(* CODESYS project EPW_3NE_slave.project
   Title: titoloSenza
   Version: 0.0.0.0
   Author: Tecnico3

Project tree, tasks and I/O mapping:
  MyController : TM241CEC24T/U, Schneider Electric, order no. TM241CEC24T/U, version 4.0.6.18
    application Application
      task MAST (cyclic, interval 10 ms, priority 15, watchdog 100 ms x 1) calls P0_Main, Clock_Encoder
      program P0_Main [SFC]: Init_active, ILS_CAN_active
      function block FB_ILS [FBD]
      function block FB_Steppers [FBD]
      Global_VAR/
        global variables GVL
        global variables GVL_HMI
        global variables GVL_IO
        global variables PersistentVars
        global variables GVL_Motion
      Symbols
      Programma/
        program P9_Slave_to_master [ST]
        program P1_Principale [ST]
        program Clock_Encoder [LD]
        program P7_Allarmi [ST]
    DI : Digital Inputs, Schneider Electric, version 4.0.6.18
        settings: IOs Usage = 3075
        input  iwDI_IW0 : WORD  // IW0
        input  Application.Potenza_Attiva : BOOL  // IW0.I4
        input  Application.UM_Abil_Vol : BOOL  // IW0.I5
        input  Application.DI_Unita_10X : BOOL  // IW0.I6
        input  ibDI_IB1 : BYTE  // IB1
    DQ : Digital Outputs, Schneider Electric, version 4.0.6.18
        settings: Outputs Usage = 15
        output Application.Y_sblocco_Carrelli : BOOL  // QW0.Q4
        output Application.Y_sblocco_Pinze : BOOL  // QW0.Q5
        unmapped channels: QW0, QB1
    Counters : Counters, Schneider Electric, version 4.0.6.18
        settings: Instance name = 'Encoder_Volantino'; B input History = 'old=-1 new=1'; A input History = 'old=-1 new=0'; Temporary Instance name = 'Encoder_Volantino'
    Pulse_Generators : Pulse Generators, Schneider Electric, version 4.0.6.18
        settings: Instance name = 'PTO_0'; REF input History = 'old=8 new=10'; B output History = 'old=-1 new=1'; A output History = 'old=-1 new=0'; Temporary Instance name = 'PTO_0'; Instance name = 'PTO_1'; REF input History = 'old=-1 new=11'; B output History = 'old=-1 new=3'; A output History = 'old=-1 new=2'; Temporary Instance name = 'PTO_1'
    Cartridge_1 : Cartridge, Schneider Electric, version 4.0.6.18
    IO_Bus : IO bus - TM3, Schneider Electric, version 4.0.6.18
    COM_Bus : COM bus, Schneider Electric, version 4.0.6.18
    Ethernet_1 : Ethernet Network, Schneider Electric, version 4.0.6.18
      EthernetIP : EthernetIP, Schneider Electric, version 3.3.0.6
          settings: Major Revision for export = 2; old params for export = [100,150,48,48]; CRC of iomapping for export = -17395944
          input  iwEthernetIP_IW0 : WORD  // IW0
          input  modo_regolazioni : BOOL  // IW0.Bit1
          input  Cancella_allarmi : BOOL  // IW0.Bit7
          input  Token : BOOL  // IW0.Bit9
          input  sblocco_carrelli : BOOL  // IW0.Bit11
          input  sblocco_pinze : BOOL  // IW0.Bit12
          input  position_setting : BOOL  // IW0.Bit14
          input  C1_enable : BOOL  // IW1.Bit0
          input  C1_home : BOOL  // IW1.Bit1
          input  C1_position : BOOL  // IW1.Bit2
          input  C1_jog : BOOL  // IW1.Bit3
          input  C1_setpos : BOOL  // IW1.Bit4
          input  C2_enable : BOOL  // IW2.Bit0
          input  C2_home : BOOL  // IW2.Bit1
          input  C2_position : BOOL  // IW2.Bit2
          input  C2_jog : BOOL  // IW2.Bit3
          input  C2_setpos : BOOL  // IW2.Bit4
          input  C3_enable : BOOL  // IW3.Bit0
          input  C3_home : BOOL  // IW3.Bit1
          input  C3_position : BOOL  // IW3.Bit2
          input  C3_jog : BOOL  // IW3.Bit3
          input  C3_setpos : BOOL  // IW3.Bit4
          input  C4_enable : BOOL  // IW4.Bit0
          input  C4_home : BOOL  // IW4.Bit1
          input  C4_position : BOOL  // IW4.Bit2
          input  C4_jog : BOOL  // IW4.Bit3
          input  C4_setpos : BOOL  // IW4.Bit4
          input  Larg_Bracci_enable : BOOL  // IW5.Bit0
          input  Larg_Bracci_home : BOOL  // IW5.Bit1
          input  Larg_Bracci_position : BOOL  // IW5.Bit2
          input  Larg_Bracci_jog : BOOL  // IW5.Bit3
          input  Larg_Bracci_setpos : BOOL  // IW5.Bit4
          input  Pinza_Sx_enable : BOOL  // IW6.Bit0
          input  Pinza_Sx_home : BOOL  // IW6.Bit1
          input  Pinza_Sx_position : BOOL  // IW6.Bit2
          input  Pinza_Sx_jog : BOOL  // IW6.Bit3
          input  Pinza_Sx_setpos : BOOL  // IW6.Bit4
          input  Pinza_Dx_enable : BOOL  // IW7.Bit0
          input  Pinza_Dx_home : BOOL  // IW7.Bit1
          input  Pinza_Dx_position : BOOL  // IW7.Bit2
          input  Pinza_Dx_jog : BOOL  // IW7.Bit3
          input  Pinza_Dx_setpos : BOOL  // IW7.Bit4
          input  iwEthernetIP_IW8 : WORD  // IW8
          input  iwEthernetIP_IW9 : WORD  // IW9
          input  iwEthernetIP_IW10 : WORD  // IW10
          input  iwEthernetIP_IW11 : WORD  // IW11
          input  iwEthernetIP_IW12 : WORD  // IW12
          input  iwEthernetIP_IW13 : WORD  // IW13
          input  iwEthernetIP_IW14 : WORD  // IW14
          input  iwEthernetIP_IW15 : WORD  // IW15
          input  Target_pos_Carrello_1 : WORD  // IW16
          input  Target_pos_Carrello_2 : WORD  // IW17
          input  Target_pos_Carrello_3 : WORD  // IW18
          input  Target_pos_Carrello_4 : WORD  // IW19
          input  Target_pos_Larg_Bracci : WORD  // IW20
          input  Target_pos_Pinza_Sx : WORD  // IW21
          input  Target_pos_Pinza_Dx : WORD  // IW22
          output PB_Abil_Vol : BOOL  // QW0.Bit5
          output Reverse_Token : BOOL  // QW0.Bit9
          output C1_errore : BOOL  // QW1.Bit0
          output C1_referenced : BOOL  // QW1.Bit1
          output C1_done_abs : BOOL  // QW1.Bit2
          output C1_done_home : BOOL  // QW1.Bit3
          output C1_done_mvadd : BOOL  // QW1.Bit4
          output C1_done_setpos : BOOL  // QW1.Bit5
          output C1_in_position : BOOL  // QW1.Bit6
          output C2_errore : BOOL  // QW2.Bit0
          output C2_referenced : BOOL  // QW2.Bit1
          output C2_done_abs : BOOL  // QW2.Bit2
          output C2_done_home : BOOL  // QW2.Bit3
          output C2_done_mvadd : BOOL  // QW2.Bit4
          output C2_done_setpos : BOOL  // QW2.Bit5
          output C2_in_position : BOOL  // QW2.Bit6
          output C3_errore : BOOL  // QW3.Bit0
          output C3_referenced : BOOL  // QW3.Bit1
          output C3_done_abs : BOOL  // QW3.Bit2
          output C3_done_home : BOOL  // QW3.Bit3
          output C3_done_mvadd : BOOL  // QW3.Bit4
          output C3_done_setpos : BOOL  // QW3.Bit5
          output C3_in_position : BOOL  // QW3.Bit6
          output C4_errore : BOOL  // QW4.Bit0
          output C4_referenced : BOOL  // QW4.Bit1
          output C4_done_abs : BOOL  // QW4.Bit2
          output C4_done_home : BOOL  // QW4.Bit3
          output C4_done_mvadd : BOOL  // QW4.Bit4
          output C4_done_setpos : BOOL  // QW4.Bit5
          output C4_in_position : BOOL  // QW4.Bit6
          output L_br_errore : BOOL  // QW5.Bit0
          output L_br_referenced : BOOL  // QW5.Bit1
          output L_br_done_abs : BOOL  // QW5.Bit2
          output L_br_done_home : BOOL  // QW5.Bit3
          output L_br_done_mvadd : BOOL  // QW5.Bit4
          output L_br_done_setpos : BOOL  // QW5.Bit5
          output L_br_in_position : BOOL  // QW5.Bit6
          output Pinza_sx_errore : BOOL  // QW6.Bit0
          output Pinza_sx_referenced : BOOL  // QW6.Bit1
          output Pinza_sx_done_abs : BOOL  // QW6.Bit2
          output Pinza_sx_done_home : BOOL  // QW6.Bit3
          output Pinza_sx_done_mvadd : BOOL  // QW6.Bit4
          output Pinza_sx_done_setpos : BOOL  // QW6.Bit5
          output Pinza_Sx_in_position : BOOL  // QW6.Bit6
          output Pinza_dx_errore : BOOL  // QW7.Bit0
          output Pinza_dx_referenced : BOOL  // QW7.Bit1
          output Pinza_dx_done_abs : BOOL  // QW7.Bit2
          output Pinza_dx_done_home : BOOL  // QW7.Bit3
          output Pinza_dx_done_mvadd : BOOL  // QW7.Bit4
          output Pinza_dx_done_setpos : BOOL  // QW7.Bit5
          output Pinza_Dx_in_position : BOOL  // QW7.Bit6
          output Fault_Carrello_1 : WORD  // QW8
          output Fault_Carrello_2 : WORD  // QW9
          output Fault_Carrello_3 : WORD  // QW10
          output Fault_Carrello_4 : WORD  // QW11
          output Fault_Larg_Bracci : WORD  // QW12
          output Fault_Pinza_Sx : WORD  // QW13
          output Fault_Pinza_Dx : WORD  // QW14
          output Actual_Position_Carrello_1 : WORD  // QW16
          output Actual_Position_Carrello_2 : WORD  // QW17
          output Actual_Position_Carrello_3 : WORD  // QW18
          output Actual_Position_Carrello_4 : WORD  // QW19
          output Actual_Position_Larg_Bracci : WORD  // QW20
          output Actual_Position_Pinza_Sx : WORD  // QW21
          output Actual_Position_Pinza_Dx : WORD  // QW22
          output Actual_Position_Volantino : WORD  // QW23
          unmapped channels: IW1, IW2, IW3, IW4, IW5, IW6, IW7, IW23, QW0, QW1, QW2, QW3, QW4, QW5, QW6, QW7, QW15
    Serial_Line_1 : Serial line, Schneider Electric, version 4.0.6.18
      SoMachine_Network_Manager : SoMachine-Network Manager, Schneider Electric, version 4.0.0.2
    Serial_Line_2 : Serial line, Schneider Electric, version 4.0.6.18
      Modbus_Manager : Modbus Manager, Schneider Electric, version 4.0.0.2
    CAN_1 : CANopen bus, Schneider Electric, version 4.0.6.18
      CANopen_Performance : CANopen Performance, Schneider Electric, order no. 1806, version 3.0.1.24
          settings: ConfigVersion = 50659584
        ILS_Carrello_1 : Lexium ILS, Schneider Electric, order no. 1, version 3.2.1.0
            settings: General Options.Optional Device = TRUE; NODEIDSAVED = 1; SDO Timeout = 1000000; Explicit Deactivate PDOs = FALSE; EXPERTSETTINGS = False; Nodeguarding.Guard Time = 200 ms; Nodeguarding.Life Time Factor = 2; PDO 16#1803.COBID = 16#0481; pdo4_driveCtrl.Subindex = 16#01; pdo4_modeCtrl.Subindex = 16#02; pdo4_Ref16.Subindex = 16#05; pdo4_Ref32.Subindex = 16#06; pdo4_driveStat.Subindex = 16#04; pdo4_modeStat.Subindex = 16#03; pdo4_Act8.Subindex = 16#07; pdo4_Act32.Subindex = 16#08; SDO List.Set Guardtime.Index = 16#100C; SDO List.Set Guardtime.Subindex = 16#00; SDO List.Set Guardtime.Value = 16#000000C8; SDO List.Set Guardtime.Size = 16; SDO List.Set Guardtime.AbortIfError = FALSE; SDO List.Set Guardtime.JumpToLine = FALSE; SDO List.Set Guardtime.Line = 0; SDO List.Set Lifetime.Index = 16#100D; SDO List.Set Lifetime.Subindex = 16#00; SDO List.Set Lifetime.Value = 16#00000002; SDO List.Set Lifetime.Size = 8; SDO List.Set Lifetime.AbortIfError = FALSE; SDO List.Set Lifetime.JumpToLine = FALSE; SDO List.Set Lifetime.Line = 0; SDO List.Disable PDO.Index = 16#1803; SDO List.Disable PDO.Subindex = 16#01; SDO List.Disable PDO.Value = 16#80000481; SDO List.Disable PDO.Size = 32; SDO List.Disable PDO.AbortIfError = FALSE; SDO List.Disable PDO.JumpToLine = FALSE; SDO List.Disable PDO.Line = 0; SDO List.Set transmission type.Index = 16#1803; SDO List.Set transmission type.Subindex = 16#02; SDO List.Set transmission type.Value = 16#FE;
              SDO List.Set transmission type.Size = 8; SDO List.Set transmission type.AbortIfError = FALSE; SDO List.Set transmission type.JumpToLine = FALSE; SDO List.Set transmission type.Line = 0; SDO List.Set inhibit time.Index = 16#1803; SDO List.Set inhibit time.Subindex = 16#03; SDO List.Set inhibit time.Value = 16#0064; SDO List.Set inhibit time.Size = 16; SDO List.Set inhibit time.AbortIfError = FALSE; SDO List.Set inhibit time.JumpToLine = FALSE; SDO List.Set inhibit time.Line = 0; SDO List.Set event time.Index = 16#1803; SDO List.Set event time.Subindex = 16#05; SDO List.Set event time.Value = 16#0000; SDO List.Set event time.Size = 16; SDO List.Set event time.AbortIfError = FALSE; SDO List.Set event time.JumpToLine = FALSE; SDO List.Set event time.Line = 0; SDO List.Set and enable COB-ID.Index = 16#1803; SDO List.Set and enable COB-ID.Subindex = 16#01; SDO List.Set and enable COB-ID.Value = 16#00000481; SDO List.Set and enable COB-ID.Size = 32; SDO List.Set and enable COB-ID.AbortIfError = FALSE; SDO List.Set and enable COB-ID.JumpToLine = FALSE; SDO List.Set and enable COB-ID.Line = 0; SDO List.Automap SDO1.Index = 16#301E; SDO List.Automap SDO1.Subindex = 16#0A; SDO List.Automap SDO1.Value = 4294967295; SDO List.Automap SDO1.Size = 32; SDO List.Automap SDO1.AbortIfError = FALSE; SDO List.Automap SDO1.JumpToLine = FALSE; SDO List.Automap SDO1.Line = 0; ConfigVersion = 50659584
            unmapped channels: pdo4_driveCtrl, pdo4_modeCtrl, pdo4_Ref16, pdo4_Ref32, pdo4_driveStat, pdo4_modeStat, pdo4_Act8, pdo4_Act32
        ILS_Carrello_2 : Lexium ILS, Schneider Electric, order no. 1, version 3.2.1.0
            settings: General Options.Optional Device = TRUE; NODEIDSAVED = 2; SDO Timeout = 1000000; Explicit Deactivate PDOs = FALSE; EXPERTSETTINGS = FALSE; Nodeguarding.Guard Time = 200 ms; Nodeguarding.Life Time Factor = 2; Emergency-General Parameters.Emergency COBID = 16#82; PDO 16#1403.COBID = 16#40000502; PDO 16#1803.COBID = 16#0482; pdo4_driveCtrl.Subindex = 16#01; pdo4_modeCtrl.Subindex = 16#02; pdo4_Ref16.Subindex = 16#05; pdo4_Ref32.Subindex = 16#06; pdo4_driveStat.Subindex = 16#04; pdo4_modeStat.Subindex = 16#03; pdo4_Act8.Subindex = 16#07; pdo4_Act32.Subindex = 16#08; SDO List.Set Guardtime.Index = 16#100C; SDO List.Set Guardtime.Subindex = 16#00; SDO List.Set Guardtime.Value = 16#000000C8; SDO List.Set Guardtime.Size = 16; SDO List.Set Guardtime.AbortIfError = FALSE; SDO List.Set Guardtime.JumpToLine = FALSE; SDO List.Set Guardtime.Line = 0; SDO List.Set Lifetime.Index = 16#100D; SDO List.Set Lifetime.Subindex = 16#00; SDO List.Set Lifetime.Value = 16#00000002; SDO List.Set Lifetime.Size = 8; SDO List.Set Lifetime.AbortIfError = FALSE; SDO List.Set Lifetime.JumpToLine = FALSE; SDO List.Set Lifetime.Line = 0; SDO List.Disable PDO.Index = 16#1803; SDO List.Disable PDO.Subindex = 16#01; SDO List.Disable PDO.Value = 16#80000482; SDO List.Disable PDO.Size = 32; SDO List.Disable PDO.AbortIfError = FALSE; SDO List.Disable PDO.JumpToLine = FALSE; SDO List.Disable PDO.Line = 0; SDO List.Set transmission type.Index = 16#1803;
              SDO List.Set transmission type.Subindex = 16#02; SDO List.Set transmission type.Value = 16#FE; SDO List.Set transmission type.Size = 8; SDO List.Set transmission type.AbortIfError = FALSE; SDO List.Set transmission type.JumpToLine = FALSE; SDO List.Set transmission type.Line = 0; SDO List.Set inhibit time.Index = 16#1803; SDO List.Set inhibit time.Subindex = 16#03; SDO List.Set inhibit time.Value = 16#0064; SDO List.Set inhibit time.Size = 16; SDO List.Set inhibit time.AbortIfError = FALSE; SDO List.Set inhibit time.JumpToLine = FALSE; SDO List.Set inhibit time.Line = 0; SDO List.Set event time.Index = 16#1803; SDO List.Set event time.Subindex = 16#05; SDO List.Set event time.Value = 16#0000; SDO List.Set event time.Size = 16; SDO List.Set event time.AbortIfError = FALSE; SDO List.Set event time.JumpToLine = FALSE; SDO List.Set event time.Line = 0; SDO List.Set and enable COB-ID.Index = 16#1803; SDO List.Set and enable COB-ID.Subindex = 16#01; SDO List.Set and enable COB-ID.Value = 16#00000482; SDO List.Set and enable COB-ID.Size = 32; SDO List.Set and enable COB-ID.AbortIfError = FALSE; SDO List.Set and enable COB-ID.JumpToLine = FALSE; SDO List.Set and enable COB-ID.Line = 0; SDO List.Automap SDO1.Index = 16#301E; SDO List.Automap SDO1.Subindex = 16#0A; SDO List.Automap SDO1.Value = 4294967295; SDO List.Automap SDO1.Size = 32; SDO List.Automap SDO1.AbortIfError = FALSE; SDO List.Automap SDO1.JumpToLine = FALSE; SDO List.Automap SDO1.Line = 0; ConfigVersion = 50659584
            unmapped channels: pdo4_driveCtrl, pdo4_modeCtrl, pdo4_Ref16, pdo4_Ref32, pdo4_driveStat, pdo4_modeStat, pdo4_Act8, pdo4_Act32
        ILS_Carrello_3 : Lexium ILS, Schneider Electric, order no. 1, version 3.2.1.0
            settings: General Options.Optional Device = TRUE; NODEIDSAVED = 3; SDO Timeout = 1000000; Explicit Deactivate PDOs = FALSE; EXPERTSETTINGS = FALSE; Nodeguarding.Guard Time = 200 ms; Nodeguarding.Life Time Factor = 2; Emergency-General Parameters.Emergency COBID = 16#83; PDO 16#1403.COBID = 16#40000503; PDO 16#1803.COBID = 16#0483; pdo4_driveCtrl.Subindex = 16#01; pdo4_modeCtrl.Subindex = 16#02; pdo4_Ref16.Subindex = 16#05; pdo4_Ref32.Subindex = 16#06; pdo4_driveStat.Subindex = 16#04; pdo4_modeStat.Subindex = 16#03; pdo4_Act8.Subindex = 16#07; pdo4_Act32.Subindex = 16#08; SDO List.Set Guardtime.Index = 16#100C; SDO List.Set Guardtime.Subindex = 16#00; SDO List.Set Guardtime.Value = 16#000000C8; SDO List.Set Guardtime.Size = 16; SDO List.Set Guardtime.AbortIfError = FALSE; SDO List.Set Guardtime.JumpToLine = FALSE; SDO List.Set Guardtime.Line = 0; SDO List.Set Lifetime.Index = 16#100D; SDO List.Set Lifetime.Subindex = 16#00; SDO List.Set Lifetime.Value = 16#00000002; SDO List.Set Lifetime.Size = 8; SDO List.Set Lifetime.AbortIfError = FALSE; SDO List.Set Lifetime.JumpToLine = FALSE; SDO List.Set Lifetime.Line = 0; SDO List.Disable PDO.Index = 16#1803; SDO List.Disable PDO.Subindex = 16#01; SDO List.Disable PDO.Value = 16#80000483; SDO List.Disable PDO.Size = 32; SDO List.Disable PDO.AbortIfError = FALSE; SDO List.Disable PDO.JumpToLine = FALSE; SDO List.Disable PDO.Line = 0; SDO List.Set transmission type.Index = 16#1803;
              SDO List.Set transmission type.Subindex = 16#02; SDO List.Set transmission type.Value = 16#FE; SDO List.Set transmission type.Size = 8; SDO List.Set transmission type.AbortIfError = FALSE; SDO List.Set transmission type.JumpToLine = FALSE; SDO List.Set transmission type.Line = 0; SDO List.Set inhibit time.Index = 16#1803; SDO List.Set inhibit time.Subindex = 16#03; SDO List.Set inhibit time.Value = 16#0064; SDO List.Set inhibit time.Size = 16; SDO List.Set inhibit time.AbortIfError = FALSE; SDO List.Set inhibit time.JumpToLine = FALSE; SDO List.Set inhibit time.Line = 0; SDO List.Set event time.Index = 16#1803; SDO List.Set event time.Subindex = 16#05; SDO List.Set event time.Value = 16#0000; SDO List.Set event time.Size = 16; SDO List.Set event time.AbortIfError = FALSE; SDO List.Set event time.JumpToLine = FALSE; SDO List.Set event time.Line = 0; SDO List.Set and enable COB-ID.Index = 16#1803; SDO List.Set and enable COB-ID.Subindex = 16#01; SDO List.Set and enable COB-ID.Value = 16#00000483; SDO List.Set and enable COB-ID.Size = 32; SDO List.Set and enable COB-ID.AbortIfError = FALSE; SDO List.Set and enable COB-ID.JumpToLine = FALSE; SDO List.Set and enable COB-ID.Line = 0; SDO List.Automap SDO1.Index = 16#301E; SDO List.Automap SDO1.Subindex = 16#0A; SDO List.Automap SDO1.Value = 4294967295; SDO List.Automap SDO1.Size = 32; SDO List.Automap SDO1.AbortIfError = FALSE; SDO List.Automap SDO1.JumpToLine = FALSE; SDO List.Automap SDO1.Line = 0; ConfigVersion = 50659584
            unmapped channels: pdo4_driveCtrl, pdo4_modeCtrl, pdo4_Ref16, pdo4_Ref32, pdo4_driveStat, pdo4_modeStat, pdo4_Act8, pdo4_Act32
        ILS_Carrello_4 : Lexium ILS, Schneider Electric, order no. 1, version 3.2.1.0
            settings: General Options.Optional Device = TRUE; NODEIDSAVED = 4; SDO Timeout = 1000000; Explicit Deactivate PDOs = FALSE; EXPERTSETTINGS = FALSE; Nodeguarding.Guard Time = 200 ms; Nodeguarding.Life Time Factor = 2; Emergency-General Parameters.Emergency COBID = 16#84; PDO 16#1403.COBID = 16#40000504; PDO 16#1803.COBID = 16#0484; pdo4_driveCtrl.Subindex = 16#01; pdo4_modeCtrl.Subindex = 16#02; pdo4_Ref16.Subindex = 16#05; pdo4_Ref32.Subindex = 16#06; pdo4_driveStat.Subindex = 16#04; pdo4_modeStat.Subindex = 16#03; pdo4_Act8.Subindex = 16#07; pdo4_Act32.Subindex = 16#08; SDO List.Set Guardtime.Index = 16#100C; SDO List.Set Guardtime.Subindex = 16#00; SDO List.Set Guardtime.Value = 16#000000C8; SDO List.Set Guardtime.Size = 16; SDO List.Set Guardtime.AbortIfError = FALSE; SDO List.Set Guardtime.JumpToLine = FALSE; SDO List.Set Guardtime.Line = 0; SDO List.Set Lifetime.Index = 16#100D; SDO List.Set Lifetime.Subindex = 16#00; SDO List.Set Lifetime.Value = 16#00000002; SDO List.Set Lifetime.Size = 8; SDO List.Set Lifetime.AbortIfError = FALSE; SDO List.Set Lifetime.JumpToLine = FALSE; SDO List.Set Lifetime.Line = 0; SDO List.Disable PDO.Index = 16#1803; SDO List.Disable PDO.Subindex = 16#01; SDO List.Disable PDO.Value = 16#80000484; SDO List.Disable PDO.Size = 32; SDO List.Disable PDO.AbortIfError = FALSE; SDO List.Disable PDO.JumpToLine = FALSE; SDO List.Disable PDO.Line = 0; SDO List.Set transmission type.Index = 16#1803;
              SDO List.Set transmission type.Subindex = 16#02; SDO List.Set transmission type.Value = 16#FE; SDO List.Set transmission type.Size = 8; SDO List.Set transmission type.AbortIfError = FALSE; SDO List.Set transmission type.JumpToLine = FALSE; SDO List.Set transmission type.Line = 0; SDO List.Set inhibit time.Index = 16#1803; SDO List.Set inhibit time.Subindex = 16#03; SDO List.Set inhibit time.Value = 16#0064; SDO List.Set inhibit time.Size = 16; SDO List.Set inhibit time.AbortIfError = FALSE; SDO List.Set inhibit time.JumpToLine = FALSE; SDO List.Set inhibit time.Line = 0; SDO List.Set event time.Index = 16#1803; SDO List.Set event time.Subindex = 16#05; SDO List.Set event time.Value = 16#0000; SDO List.Set event time.Size = 16; SDO List.Set event time.AbortIfError = FALSE; SDO List.Set event time.JumpToLine = FALSE; SDO List.Set event time.Line = 0; SDO List.Set and enable COB-ID.Index = 16#1803; SDO List.Set and enable COB-ID.Subindex = 16#01; SDO List.Set and enable COB-ID.Value = 16#00000484; SDO List.Set and enable COB-ID.Size = 32; SDO List.Set and enable COB-ID.AbortIfError = FALSE; SDO List.Set and enable COB-ID.JumpToLine = FALSE; SDO List.Set and enable COB-ID.Line = 0; SDO List.Automap SDO1.Index = 16#301E; SDO List.Automap SDO1.Subindex = 16#0A; SDO List.Automap SDO1.Value = 4294967295; SDO List.Automap SDO1.Size = 32; SDO List.Automap SDO1.AbortIfError = FALSE; SDO List.Automap SDO1.JumpToLine = FALSE; SDO List.Automap SDO1.Line = 0; ConfigVersion = 50659584
            unmapped channels: pdo4_driveCtrl, pdo4_modeCtrl, pdo4_Ref16, pdo4_Ref32, pdo4_driveStat, pdo4_modeStat, pdo4_Act8, pdo4_Act32
        ILS_Larg_Bracci : Lexium ILS, Schneider Electric, order no. 1, version 3.2.1.0
            settings: General Options.Optional Device = TRUE; NODEIDSAVED = 5; SDO Timeout = 1000000; Explicit Deactivate PDOs = FALSE; EXPERTSETTINGS = FALSE; Nodeguarding.Guard Time = 200 ms; Nodeguarding.Life Time Factor = 2; Emergency-General Parameters.Emergency COBID = 16#85; PDO 16#1403.COBID = 16#40000505; PDO 16#1803.COBID = 16#0485; pdo4_driveCtrl.Subindex = 16#01; pdo4_modeCtrl.Subindex = 16#02; pdo4_Ref16.Subindex = 16#05; pdo4_Ref32.Subindex = 16#06; pdo4_driveStat.Subindex = 16#04; pdo4_modeStat.Subindex = 16#03; pdo4_Act8.Subindex = 16#07; pdo4_Act32.Subindex = 16#08; SDO List.Set Guardtime.Index = 16#100C; SDO List.Set Guardtime.Subindex = 16#00; SDO List.Set Guardtime.Value = 16#000000C8; SDO List.Set Guardtime.Size = 16; SDO List.Set Guardtime.AbortIfError = FALSE; SDO List.Set Guardtime.JumpToLine = FALSE; SDO List.Set Guardtime.Line = 0; SDO List.Set Lifetime.Index = 16#100D; SDO List.Set Lifetime.Subindex = 16#00; SDO List.Set Lifetime.Value = 16#00000002; SDO List.Set Lifetime.Size = 8; SDO List.Set Lifetime.AbortIfError = FALSE; SDO List.Set Lifetime.JumpToLine = FALSE; SDO List.Set Lifetime.Line = 0; SDO List.Disable PDO.Index = 16#1803; SDO List.Disable PDO.Subindex = 16#01; SDO List.Disable PDO.Value = 16#80000485; SDO List.Disable PDO.Size = 32; SDO List.Disable PDO.AbortIfError = FALSE; SDO List.Disable PDO.JumpToLine = FALSE; SDO List.Disable PDO.Line = 0; SDO List.Set transmission type.Index = 16#1803;
              SDO List.Set transmission type.Subindex = 16#02; SDO List.Set transmission type.Value = 16#FE; SDO List.Set transmission type.Size = 8; SDO List.Set transmission type.AbortIfError = FALSE; SDO List.Set transmission type.JumpToLine = FALSE; SDO List.Set transmission type.Line = 0; SDO List.Set inhibit time.Index = 16#1803; SDO List.Set inhibit time.Subindex = 16#03; SDO List.Set inhibit time.Value = 16#0064; SDO List.Set inhibit time.Size = 16; SDO List.Set inhibit time.AbortIfError = FALSE; SDO List.Set inhibit time.JumpToLine = FALSE; SDO List.Set inhibit time.Line = 0; SDO List.Set event time.Index = 16#1803; SDO List.Set event time.Subindex = 16#05; SDO List.Set event time.Value = 16#0000; SDO List.Set event time.Size = 16; SDO List.Set event time.AbortIfError = FALSE; SDO List.Set event time.JumpToLine = FALSE; SDO List.Set event time.Line = 0; SDO List.Set and enable COB-ID.Index = 16#1803; SDO List.Set and enable COB-ID.Subindex = 16#01; SDO List.Set and enable COB-ID.Value = 16#00000485; SDO List.Set and enable COB-ID.Size = 32; SDO List.Set and enable COB-ID.AbortIfError = FALSE; SDO List.Set and enable COB-ID.JumpToLine = FALSE; SDO List.Set and enable COB-ID.Line = 0; SDO List.Automap SDO1.Index = 16#301E; SDO List.Automap SDO1.Subindex = 16#0A; SDO List.Automap SDO1.Value = 4294967295; SDO List.Automap SDO1.Size = 32; SDO List.Automap SDO1.AbortIfError = FALSE; SDO List.Automap SDO1.JumpToLine = FALSE; SDO List.Automap SDO1.Line = 0; ConfigVersion = 50659584
            unmapped channels: pdo4_driveCtrl, pdo4_modeCtrl, pdo4_Ref16, pdo4_Ref32, pdo4_driveStat, pdo4_modeStat, pdo4_Act8, pdo4_Act32
        ILS_Pinza_Sx : Lexium ILS, Schneider Electric, order no. 1, version 3.2.1.0
            settings: General Options.Optional Device = TRUE; NODEIDSAVED = 6; SDO Timeout = 1000000; Explicit Deactivate PDOs = FALSE; EXPERTSETTINGS = FALSE; Nodeguarding.Guard Time = 200 ms; Nodeguarding.Life Time Factor = 2; Emergency-General Parameters.Emergency COBID = 16#86; PDO 16#1403.COBID = 16#40000506; PDO 16#1803.COBID = 16#0486; pdo4_driveCtrl.Subindex = 16#01; pdo4_modeCtrl.Subindex = 16#02; pdo4_Ref16.Subindex = 16#05; pdo4_Ref32.Subindex = 16#06; pdo4_driveStat.Subindex = 16#04; pdo4_modeStat.Subindex = 16#03; pdo4_Act8.Subindex = 16#07; pdo4_Act32.Subindex = 16#08; SDO List.Set Guardtime.Index = 16#100C; SDO List.Set Guardtime.Subindex = 16#00; SDO List.Set Guardtime.Value = 16#000000C8; SDO List.Set Guardtime.Size = 16; SDO List.Set Guardtime.AbortIfError = FALSE; SDO List.Set Guardtime.JumpToLine = FALSE; SDO List.Set Guardtime.Line = 0; SDO List.Set Lifetime.Index = 16#100D; SDO List.Set Lifetime.Subindex = 16#00; SDO List.Set Lifetime.Value = 16#00000002; SDO List.Set Lifetime.Size = 8; SDO List.Set Lifetime.AbortIfError = FALSE; SDO List.Set Lifetime.JumpToLine = FALSE; SDO List.Set Lifetime.Line = 0; SDO List.Disable PDO.Index = 16#1803; SDO List.Disable PDO.Subindex = 16#01; SDO List.Disable PDO.Value = 16#80000486; SDO List.Disable PDO.Size = 32; SDO List.Disable PDO.AbortIfError = FALSE; SDO List.Disable PDO.JumpToLine = FALSE; SDO List.Disable PDO.Line = 0; SDO List.Set transmission type.Index = 16#1803;
              SDO List.Set transmission type.Subindex = 16#02; SDO List.Set transmission type.Value = 16#FE; SDO List.Set transmission type.Size = 8; SDO List.Set transmission type.AbortIfError = FALSE; SDO List.Set transmission type.JumpToLine = FALSE; SDO List.Set transmission type.Line = 0; SDO List.Set inhibit time.Index = 16#1803; SDO List.Set inhibit time.Subindex = 16#03; SDO List.Set inhibit time.Value = 16#0064; SDO List.Set inhibit time.Size = 16; SDO List.Set inhibit time.AbortIfError = FALSE; SDO List.Set inhibit time.JumpToLine = FALSE; SDO List.Set inhibit time.Line = 0; SDO List.Set event time.Index = 16#1803; SDO List.Set event time.Subindex = 16#05; SDO List.Set event time.Value = 16#0000; SDO List.Set event time.Size = 16; SDO List.Set event time.AbortIfError = FALSE; SDO List.Set event time.JumpToLine = FALSE; SDO List.Set event time.Line = 0; SDO List.Set and enable COB-ID.Index = 16#1803; SDO List.Set and enable COB-ID.Subindex = 16#01; SDO List.Set and enable COB-ID.Value = 16#00000486; SDO List.Set and enable COB-ID.Size = 32; SDO List.Set and enable COB-ID.AbortIfError = FALSE; SDO List.Set and enable COB-ID.JumpToLine = FALSE; SDO List.Set and enable COB-ID.Line = 0; SDO List.Automap SDO1.Index = 16#301E; SDO List.Automap SDO1.Subindex = 16#0A; SDO List.Automap SDO1.Value = 4294967295; SDO List.Automap SDO1.Size = 32; SDO List.Automap SDO1.AbortIfError = FALSE; SDO List.Automap SDO1.JumpToLine = FALSE; SDO List.Automap SDO1.Line = 0; ConfigVersion = 50659584
            unmapped channels: pdo4_driveCtrl, pdo4_modeCtrl, pdo4_Ref16, pdo4_Ref32, pdo4_driveStat, pdo4_modeStat, pdo4_Act8, pdo4_Act32
        ILS_Pinza_Dx : Lexium ILS, Schneider Electric, order no. 1, version 3.2.1.0
            settings: General Options.Optional Device = TRUE; NODEIDSAVED = 7; SDO Timeout = 1000000; Explicit Deactivate PDOs = FALSE; EXPERTSETTINGS = FALSE; Nodeguarding.Guard Time = 200 ms; Nodeguarding.Life Time Factor = 2; Emergency-General Parameters.Emergency COBID = 16#87; PDO 16#1403.COBID = 16#40000507; PDO 16#1803.COBID = 16#0487; pdo4_driveCtrl.Subindex = 16#01; pdo4_modeCtrl.Subindex = 16#02; pdo4_Ref16.Subindex = 16#05; pdo4_Ref32.Subindex = 16#06; pdo4_driveStat.Subindex = 16#04; pdo4_modeStat.Subindex = 16#03; pdo4_Act8.Subindex = 16#07; pdo4_Act32.Subindex = 16#08; SDO List.Set Guardtime.Index = 16#100C; SDO List.Set Guardtime.Subindex = 16#00; SDO List.Set Guardtime.Value = 16#000000C8; SDO List.Set Guardtime.Size = 16; SDO List.Set Guardtime.AbortIfError = FALSE; SDO List.Set Guardtime.JumpToLine = FALSE; SDO List.Set Guardtime.Line = 0; SDO List.Set Lifetime.Index = 16#100D; SDO List.Set Lifetime.Subindex = 16#00; SDO List.Set Lifetime.Value = 16#00000002; SDO List.Set Lifetime.Size = 8; SDO List.Set Lifetime.AbortIfError = FALSE; SDO List.Set Lifetime.JumpToLine = FALSE; SDO List.Set Lifetime.Line = 0; SDO List.Disable PDO.Index = 16#1803; SDO List.Disable PDO.Subindex = 16#01; SDO List.Disable PDO.Value = 16#80000487; SDO List.Disable PDO.Size = 32; SDO List.Disable PDO.AbortIfError = FALSE; SDO List.Disable PDO.JumpToLine = FALSE; SDO List.Disable PDO.Line = 0; SDO List.Set transmission type.Index = 16#1803;
              SDO List.Set transmission type.Subindex = 16#02; SDO List.Set transmission type.Value = 16#FE; SDO List.Set transmission type.Size = 8; SDO List.Set transmission type.AbortIfError = FALSE; SDO List.Set transmission type.JumpToLine = FALSE; SDO List.Set transmission type.Line = 0; SDO List.Set inhibit time.Index = 16#1803; SDO List.Set inhibit time.Subindex = 16#03; SDO List.Set inhibit time.Value = 16#0064; SDO List.Set inhibit time.Size = 16; SDO List.Set inhibit time.AbortIfError = FALSE; SDO List.Set inhibit time.JumpToLine = FALSE; SDO List.Set inhibit time.Line = 0; SDO List.Set event time.Index = 16#1803; SDO List.Set event time.Subindex = 16#05; SDO List.Set event time.Value = 16#0000; SDO List.Set event time.Size = 16; SDO List.Set event time.AbortIfError = FALSE; SDO List.Set event time.JumpToLine = FALSE; SDO List.Set event time.Line = 0; SDO List.Set and enable COB-ID.Index = 16#1803; SDO List.Set and enable COB-ID.Subindex = 16#01; SDO List.Set and enable COB-ID.Value = 16#00000487; SDO List.Set and enable COB-ID.Size = 32; SDO List.Set and enable COB-ID.AbortIfError = FALSE; SDO List.Set and enable COB-ID.JumpToLine = FALSE; SDO List.Set and enable COB-ID.Line = 0; SDO List.Automap SDO1.Index = 16#301E; SDO List.Automap SDO1.Subindex = 16#0A; SDO List.Automap SDO1.Value = 4294967295; SDO List.Automap SDO1.Size = 32; SDO List.Automap SDO1.AbortIfError = FALSE; SDO List.Automap SDO1.JumpToLine = FALSE; SDO List.Automap SDO1.Line = 0; ConfigVersion = 50659584
            unmapped channels: pdo4_driveCtrl, pdo4_modeCtrl, pdo4_Ref16, pdo4_Ref32, pdo4_driveStat, pdo4_modeStat, pdo4_Act8, pdo4_Act32
*)

// MyController/Application/Global_VAR/GVL
VAR_GLOBAL
	Power_Carrello_1: BOOL;
	Stop_Carrello_1: BOOL;
	Reset_Carrello_1: BOOL;
	Home_Carrello_1: BOOL;
	Home_Pos_Carrello_1: DINT;
	HomingMode_Carrello_1: UINT;
	VHome_Carrello_1: UINT;
	VoutHome_Carrello_1: UINT;
	PoutHome_Carrello_1: DINT;
	PDisHome_Carrello_1: DINT;
	Forward_Jog_Carrello_1: BOOL;
	Backward_Jog_Carrello_1: BOOL;
	Fast_Jog_Carrello_1: BOOL;
	Tip_Jog_Carrello_1: UINT;
	Wait_Jog_Carrello_1: UINT;
	VSlow_Jog_Carrello_1: INT;
	VFast_Jog_Carrello_1: INT;
	Abs_Carrello_1: BOOL;
	Pos_Abs_Carrello_1: DINT;
	Vel_Abs_Carrello_1: INT;
	Add_Carrello_1: BOOL;
	Distance_Add_Carrello_1: DINT;
	Vel_Add_Carrello_1: INT;
	Referenced_Carrello_1: BOOL;
	StandStill_Carrello_1: BOOL;
	Done_Abs_Carrello_1: BOOL;
	Done_MAdd_Carrello_1: BOOL;
	ErrorID_Carrello_1: WORD;
	Error_Carrello_1: BOOL;
	Power_Carrello_2: BOOL;
	Stop_Carrello_2: BOOL;
	Reset_Carrello_2: BOOL;
	Home_Carrello_2: BOOL;
	Home_Pos_Carrello_2: DINT;
	HomingMode_Carrello_2: UINT;
	VHome_Carrello_2: UINT;
	VoutHome_Carrello_2: UINT;
	PoutHome_Carrello_2: DINT;
	PDisHome_Carrello_2: DINT;
	Forward_Jog_Carrello_2: BOOL;
	Backward_Jog_Carrello_2: BOOL;
	Fast_Jog_Carrello_2: BOOL;
	Tip_Jog_Carrello_2: UINT;
	Wait_Jog_Carrello_2: UINT;
	VSlow_Jog_Carrello_2: INT;
	VFast_Jog_Carrello_2: INT;
	Abs_Carrello_2: BOOL;
	Pos_Abs_Carrello_2: DINT;
	Vel_Abs_Carrello_2: INT;
	Add_Carrello_2: BOOL;
	Distance_Add_Carrello_2: DINT;
	Vel_Add_Carrello_2: INT;
	Referenced_Carrello_2: BOOL;
	StandStill_Carrello_2: BOOL;
	Done_Abs_Carrello_2: BOOL;
	Done_MAdd_Carrello_2: BOOL;
	ErrorID_Carrello_2: WORD;
	Error_Carrello_2: BOOL;
	Power_Carrello_3: BOOL;
	Stop_Carrello_3: BOOL;
	Reset_Carrello_3: BOOL;
	Home_Carrello_3: BOOL;
	Home_Pos_Carrello_3: DINT;
	HomingMode_Carrello_3: UINT;
	VHome_Carrello_3: UINT;
	VoutHome_Carrello_3: UINT;
	PoutHome_Carrello_3: DINT;
	PDisHome_Carrello_3: DINT;
	Forward_Jog_Carrello_3: BOOL;
	Backward_Jog_Carrello_3: BOOL;
	Fast_Jog_Carrello_3: BOOL;
	Tip_Jog_Carrello_3: UINT;
	Wait_Jog_Carrello_3: UINT;
	VSlow_Jog_Carrello_3: INT;
	VFast_Jog_Carrello_3: INT;
	Abs_Carrello_3: BOOL;
	Pos_Abs_Carrello_3: DINT;
	Vel_Abs_Carrello_3: INT;
	Add_Carrello_3: BOOL;
	Distance_Add_Carrello_3: DINT;
	Vel_Add_Carrello_3: INT;
	Referenced_Carrello_3: BOOL;
	StandStill_Carrello_3: BOOL;
	Done_Abs_Carrello_3: BOOL;
	Done_MAdd_Carrello_3: BOOL;
	ErrorID_Carrello_3: WORD;
	Error_Carrello_3: BOOL;
	Power_Carrello_4: BOOL;
	Stop_Carrello_4: BOOL;
	Reset_Carrello_4: BOOL;
	Home_Carrello_4: BOOL;
	Home_Pos_Carrello_4: DINT;
	HomingMode_Carrello_4: UINT;
	VHome_Carrello_4: UINT;
	VoutHome_Carrello_4: UINT;
	PoutHome_Carrello_4: DINT;
	PDisHome_Carrello_4: DINT;
	Forward_Jog_Carrello_4: BOOL;
	Backwad_Jog_Carrello_4: BOOL;
	Fast_Jog_Carrello_4: BOOL;
	Tip_Jog_Carrello_4: UINT;
	Wait_Jog_Carrello_4: UINT;
	VSlow_Jog_Carrello_4: INT;
	VFast_Jog_Carrello_4: INT;
	Abs_Carrello_4: BOOL;
	Pos_Abs_Carrello_4: DINT;
	Vel_Abs_Carrello_4: INT;
	Add_Carrello_4: BOOL;
	Distance_Add_Carrello_4: DINT;
	Vel_Add_Carrello_4: INT;
	Referenced_Carrello_4: BOOL;
	StandStill_Carrello_4: BOOL;
	Done_Abs_Carrello_4: BOOL;
	Done_MAdd_Carrello_4: BOOL;
	ErrorID_Carrello_4: WORD;
	Error_Carrello_4: BOOL;
	Power_Larg_Bracci: BOOL;
	Stop_Larg_Bracci: BOOL;
	Reset_Larg_Bracci: BOOL;
	Home_Larg_Bracci: BOOL;
	Home_Pos_Larg_Bracci: DINT;
	HomingMode_Larg_Bracci: UINT;
	VHome_Larg_Bracci: UINT;
	VoutHome_Larg_Bracci: UINT;
	PoutHome_Larg_Bracci: DINT;
	PDisHome_Larg_Bracci: DINT;
	Forward_Jog_Larg_Bracci: BOOL;
	Backward_Jog_Larg_Bracci: BOOL;
	Fast_Jog_Larg_Bracci: BOOL;
	Tip_Jog_Larg_Bracci: UINT;
	Wait_Jog_Larg_Bracci: UINT;
	VSlow_Jog_Larg_Bracci: INT;
	VFast_Jog_Larg_Bracci: INT;
	Abs_Larg_Bracci: BOOL;
	Pos_Abs_Larg_Bracci: DINT;
	Vel_Abs_Larg_Bracci: INT;
	Add_Larg_Bracci: BOOL;
	Distance_Add_Larg_Bracci: DINT;
	Vel_Add_Larg_Bracci: INT;
	Referenced_Larg_Bracci: BOOL;
	StandStill_Larg_Bracci: BOOL;
	Done_Abs_Larg_Bracci: BOOL;
	Done_MAdd_Larg_Bracci: BOOL;
	ErrorID_Larg_Bracci: WORD;
	Error_Larg_Bracci: BOOL;
	Power_Pinza_Sx: BOOL;
	Stop_Pinza_Sx: BOOL;
	Reset_Pinza_Sx: BOOL;
	Home_Pinza_Sx: BOOL;
	Home_Pos_Pinza_Sx: DINT;
	HomingMode_Pinza_Sx: UINT;
	VHome_Pinza_Sx: UINT;
	VoutHome_Pinza_Sx: UINT;
	PoutHome_Pinza_Sx: DINT;
	PDisHome_Pinza_Sx: DINT;
	Forward_Jog_Pinza_Sx: BOOL;
	Backward_Jog_Pinza_Sx: BOOL;
	Fast_Jog_Pinza_Sx: BOOL;
	Tip_Jog_Pinza_Sx: UINT;
	Wait_Jog_Pinza_Sx: UINT;
	VSlow_Jog_Pinza_Sx: INT;
	VFast_Jog_Pinza_Sx: INT;
	Abs_Pinza_Sx: BOOL;
	Pos_Abs_Pinza_Sx: DINT;
	Vel_Abs_Pinza_Sx: INT;
	Add_Pinza_Sx: BOOL;
	Distance_Add_Pinza_Sx: DINT;
	Vel_Add_Pinza_Sx: INT;
	Referenced_Pinza_Sx: BOOL;
	StandStill_Pinza_Sx: BOOL;
	Done_Abs_Pinza_Sx: BOOL;
	Done_MAdd_Pinza_Sx: BOOL;
	ErrorID_Pinza_Sx: WORD;
	Error_Pinza_Sx: BOOL;
	Power_Pinza_Dx: BOOL;
	Stop_Pinza_Dx: BOOL;
	Reset_Pinza_Dx: BOOL;
	Home_Pinza_Dx: BOOL;
	Home_Pos_Pinza_Dx: DINT;
	HomingMode_Pinza_Dx: UINT;
	VHome_Pinza_Dx: UINT;
	VoutHome_Pinza_Dx: UINT;
	PoutHome_Pinza_Dx: DINT;
	PDisHome_Pinza_Dx: DINT;
	Forward_Jog_Pinza_Dx: BOOL;
	Backward_Jog_Pinza_Dx: BOOL;
	Fast_Jog_Pinza_Dx: BOOL;
	Tip_Jog_Pinza_Dx: UINT;
	Wait_Jog_Pinza_Dx: UINT;
	VSlow_Jog_Pinza_Dx: INT;
	VFast_Jog_Pinza_Dx: INT;
	Abs_Pinza_Dx: BOOL;
	Pos_Abs_Pinza_Dx: DINT;
	Vel_Abs_Pinza_Dx: INT;
	Add_Pinza_Dx: BOOL;
	Distance_Add_Pinza_Dx: DINT;
	Vel_Add_Pinza_Dx: INT;
	Referenced_Pinza_Dx: BOOL;
	StandStill_Pinza_Dx: BOOL;
	Done_Abs_Pinza_Dx: BOOL;
	Done_MAdd_Pinza_Dx: BOOL;
	ErrorID_Pinza_Dx: WORD;
	Error_Pinza_Dx: BOOL;
	Power_PTO_0: BOOL;
	DriveReady_Power_PTO_0: BOOL;
	Limp_Power_PTO_0: BOOL;
	LimN_Power_PTO_0: BOOL;
	Reset_PTO_0: BOOL;
	Stop_PTO_0: BOOL;
	Decel_Stop_PTO_0: DINT;
	JerkRatio_Stop_PTO_0: INT;
	ReadAxis_Error_PTO_0: BOOL;
	Home_PTO_0: BOOL;
	Mode_Home_PTO_0: PTO_HOMING_MODE;
	Position_Home_PTO_0: DINT;
	Direction_Home_PTO_0: MC_DIRECTION;
	LowLev_Home_PTO_0: DINT;
	LowLev_Home_PTO_1: INT;
	High_Vel_Home_PTO_0: INT;
	High_Vel_Home_PTO_1: INT;
	Accel_Home_PTO_0: DINT;
	Decel_Home_PTO_0: DINT;
	Offset_Home_PTO_0: DINT;
	JerkRatio_Home_PTO_0: INT;
	MoveAbsolute_PTO_0: BOOL;
	Position_MoveAbs_PTO_0: DINT;
	Vel_MoveAbs_PTO_0: DINT;
	Accel_MoveAbs_PTO_0: DINT;
	Decel_MoveAbs_PTO_0: DINT;
	BufferMode_MoveAbs_PTO_0: MC_BUFFER_MODE;
	JerkRatio_MoveAbs_PTO_0: INT;
	MoveRelative_PTO_0: BOOL;
	Distance_MoveRelative_PTO_0: DINT;
	Accel_MoveRelative_PTO_0: DINT;
	Decel_MoveRelative_PTO_0: DINT;
	BufferMode_MoveRelative_PTO_0: MC_BUFFER_MODE;
	JerkRatio_MoveRelative_PTO_0: INT;
	Vel_MoveRelative_PTO_0: DINT;
	ReadActualPosition_PTO_0: BOOL;
	ReadActualVelocity_PTO_0: BOOL;
	SetPosition_PTO_0: BOOL;
	ReadStatus_PTO_0: BOOL;
	Power_PTO_1: BOOL;
	DriveReady_Power_PTO_1: BOOL;
	LimP_Power_PTO_1: BOOL;
	LimN_Power_PTO_1: BOOL;
	Reset_PTO_1: BOOL;
	Stop_PTO_1: BOOL;
	Decel_Stop_PTO_1: DINT;
	JerkRatio_Stop_PTO_1: INT;
	ReadAxisError_PTO_1: BOOL;
	Home_PTO_1: BOOL;
	Mode_Home_PTO_1: PTO_HOMING_MODE;
	Position_Home_PTO_1: DINT;
	Direction_Home_PTO_1: MC_DIRECTION;
	HighVel_Home_PTO_1: DINT;
	LowVel_Home_PTO_1: DINT;
	Accel_Home_PTO_1: DINT;
	Decel_Home_PTO_1: DINT;
	Offset_Home_PTO_1: DINT;
	JerkRatio_Home_PTO_1: INT;
	MoveAbsolute_PTO_1: BOOL;
	Position_MoveAbs_PTO_1: DINT;
	Vel_MoveAbs_PTO_1: DINT;
	Accel_MoveAbs_PTO_1: DINT;
	Decel_MoveAbs_PTO_1: DINT;
	BufferMode_MoveAbs_PTO_1: MC_BUFFER_MODE;
	JerkRatio_MoveAbs_PTO_1: INT;
	MoveRelative_PTO_1: BOOL;
	Distance_MoveRelative_PTO_1: DINT;
	Vel_MoveRelative_PTO_1: DINT;
	Accel_MoveRelative_PTO_1: DINT;
	Decel_MoveRelative_PTO_1: DINT;
	BufferMode_MoveRelative_PTO_1: MC_BUFFER_MODE;
	JerkRatio_MoveRelative_PTO_1: INT;
	ReadActualPosition_PTO_1: BOOL;
	ReadActualVelocity_PTO_1: BOOL;
	SetPosition_PTO_1: BOOL;
	ReadStatus_PTO_1: BOOL;
	ErrorId_PTO_0: PTO_ERROR;
	StandStill_PTO_0: BOOL;
	DoneAbs_PTO_0: BOOL;
	DoneMoreRel_PTO_0: BOOL;
	Error_PTO_0: BOOL;
	ErrorId_PTO_1: PTO_ERROR;
	StandStill_PTO_1: BOOL;
	DoneAbs_PTO_1: BOOL;
	Done_MoreRel_PTO_1: BOOL;
	Error_PTO_1: BOOL;
	Read_ActPosition_Carrello_1: BOOL;
	PositionType_Carrello_1: INT;
	Read_ActPosition_Carello_2: BOOL;
	PositionType_Carrello_2: INT;
	Read_ActPosition_Carrello_3: BOOL;
	PositionType_Carrello_3: INT;
	Read_ActPosition_Carello_4: BOOL;
	PositionType_Carrello_4: INT;
	Read_ActPosition_Larg_Bracci: BOOL;
	PositionType_Larg_Bracci: INT;
	Read_ActPosition_Pinza_Sx: BOOL;
	PositionType_Pinza_Sx: INT;
	Read_ActPosition_Pinza_Dx: BOOL;
	PositionType_Pinza_Dx: INT;
	ActPosition_Carrello_1: DINT;
	ActPosition_Carrello_2: DINT;
	ActPosition_Carrello_3: DINT;
	ActPosition_Carrello_4: DINT;
	ActPosition_Larg_Bracci: DINT;
	ActPosition_Pinza_Sx: DINT;
	ActPosition_Pinza_Dx: DINT;
	ActPosition_PTO_0: DINT;
	ActPosition_PTO_1: DINT;
	SetPosition_Carrello_1: BOOL;
	ModeSetPos_Carrello_1: BOOL;
	SetPosition_Carrello_2: BOOL;
	ModeSetPos_Carrello_2: BOOL;
	SetPosition_Carrello_3: BOOL;
	ModeSetPos_Carrello_3: BOOL;
	SetPosition_Carrello_4: BOOL;
	ModeSetPos_Carrello_4: BOOL;
	SetPosition_Larg_Bracci: BOOL;
	ModeSetPos_Larg_Bracci: BOOL;
	SetPosition_Pinza_Sx: BOOL;
	ModeSetPos_Pinza_Sx: BOOL;
	SetPosition_Pinza_Dx: BOOL;
	ModeSetPos_Pinza_Dx: BOOL;
	
	BusyAdd_Larg_Bracci:BOOL;
	
	//Formato Scatole
	M241_Largh_Max_Scat: INT; 
	M241_Largh_Min_Scat: INT;
	M241_Lungh_Max_Scat: INT;
	M241_Lungh_Min_Scat: INT;
	
	BusyHome_Carrello1: BOOL;
	BusyHome_Carrello2: BOOL;
	BusyHome_Carrello3: BOOL;
	BusyHome_Carrello4: BOOL;
	BusyHome_Larg_Bracci: BOOL;
	BusyHome_Pinza_Sx: BOOL;
	BusyHome_Pinza_Dx: BOOL;
	BusySPos_Carrello1: BOOL;
	BusySPos_Carrello2: BOOL;
	BusySPos_Carrello3: BOOL;
	BusySPos_Carrello4: BOOL;
	BusySPos_Larg_Bracci: BOOL;
	BusySPos_Pinza_Sx: BOOL;
	BusySPos_Pinza_Dx: BOOL;
	BusyHome_PTO_0: BOOL;
	BusyHome_PTO_1: BOOL;
	Done_SPos_PTO_0: BOOL;
	Done_SPos_PTO_1: BOOL;
	BusyAbs_Carrello1: BOOL;
	BusyAbs_Carrello2: BOOL;
	BusyAbs_Carrello3: BOOL;
	BusyAbs_Carrello4: BOOL;
	BusyAbs_Larg_Bracci: BOOL;
	BusyAbs_Pinza_Sx: BOOL;
	BusyAbs_Pinza_Dx: BOOL;
	BusyAbs_PTO_0: BOOL;
	BusyAbs_PTO_1: BOOL;
	
	Px_Home_PTO_0: BOOL; //Sensore Proximity Centratore 1
	Px_Home_PTO_1: BOOL; //Sensore Proximity Centratore 2
	
	DoneHome_PTO_0: BOOL;
	DoneHome_PTO_1: BOOL;
	BusyAdd_Carrello1: BOOL;
	BusyAdd_Carrello2: BOOL;
	BusyAdd_Carrello3: BOOL;
	BusyAdd_Carrello4: BOOL;
	BusyAdd_Pinza_Sx: BOOL;
	BusyAdd_Pinza_Dx: BOOL;
	Enc_Vol_Restart: BOOL;
	Enc_Vol_rstrt_ack: BOOL;
	Last_Encoder_Vol: DINT;
	Encoder_Vol: DINT;
	Delta_encvol: DINT;
	
	
	DoneHome_Carr1: BOOL;
	DoneHome_Carr2: BOOL;
	DoneHome_Carr3: BOOL;
	DoneHome_Carr4: BOOL;
	DoneHome_Larg_Bracci: BOOL;
	DoneHome_Pinza_Sx: BOOL;
	DoneHome_Pinza_Dx: BOOL;
	
	

	
	ck_01_s: BOOL;
	sample_clock: BOOL;
	
	Comando_globale	  :	WORD_AS_BIT;
	Comando_carrello_1: WORD_AS_BIT;
	Comando_carrello_2: WORD_AS_BIT;
	Comando_carrello_3: WORD_AS_BIT;
	Comando_carrello_4: WORD_AS_BIT;
	Comando_Larg_Bracci: WORD_AS_BIT;
	Comando_Pinza_Sx: WORD_AS_BIT;
	Comando_Pinza_Dx: WORD_AS_BIT;
	Comando_centratore_1: WORD_AS_BIT;
	Comando_centratore_2: WORD_AS_BIT;
	
//	C1_enable: 			BOOL;
//	C1_home: 			BOOL;
//	C1_position: 		BOOL;
	C1_stop_reset: 		BOOL;
//	C1_jog: 			BOOL;
	C1_attivo:		    BOOL;
//	C1_setpos:			BOOL;
	
//	C2_enable: 			BOOL;
//	C2_home: 			BOOL;
//	C2_position: 		BOOL;
	C2_stop_reset: 		BOOL;
//	C2_jog: 			BOOL;
	C2_attivo: 			BOOL;
//	C2_setpos:			BOOL;
	
//	C3_enable: 			BOOL;
//	C3_home: 			BOOL;
//	C3_position: 		BOOL;
	C3_stop_reset: 		BOOL;
//	C3_jog: 			BOOL;
	C3_attivo: 			BOOL;
//	C3_setpos:			BOOL;
	
//	C4_enable: 			BOOL;
//	C4_home: 			BOOL;
//	C4_position: 		BOOL;
	C4_stop_reset: 		BOOL;
//	C4_jog: 			BOOL;
	C4_attivo: 			BOOL;
//	C4_setpos:			BOOL;
	
//	Larg_Bracci_enable: 		BOOL;
//	Larg_Bracci_home: 			BOOL;
//	Larg_Bracci_position: 		BOOL;
	Larg_Bracci_stop_reset: 	BOOL;
//	Larg_Bracci_jog: 			BOOL;
	Larg_Bracci_attivo: 		BOOL;
//	Larg_Bracci_setpos:			BOOL;
	
//	Pinza_Sx_enable: 	BOOL;
//	Pinza_Sx_home: 		BOOL;
//	Pinza_Sx_position: 	BOOL;
	Pinza_Sx_stop_reset: 	BOOL;
//	Pinza_Sx_jog: 		BOOL;
//	Pinza_Sx_attivo: 	BOOL;
//	Pinza_Sx_setpos:	BOOL;
	
//	Pinza_Dx_enable: 	BOOL;
//	Pinza_Dx_home: 		BOOL;
//	Pinza_Dx_position: 	BOOL;
	Pinza_Dx_stop_reset: 	BOOL;
//	Pinza_Dx_jog: 		BOOL;
//	Pinza_Dx_setpos:	BOOL;
	
//	modo_regolazioni: BOOL;
//	sblocco_carrelli: BOOL;
//	sblocco_Pinze: BOOL;
//	sblocco_Larg_Bracci: BOOL;
(*	
	Target_Pos_Carrello_1: DINT;
	Target_Pos_Carrello_2: DINT;
	Target_Pos_Carrello_3: DINT;
	Target_Pos_Carrello_4: DINT;
	Target_Pos_Larg_Bracci: DINT;
	Target_Pos_Pinza_Sx: DINT;
	Target_Pos_Pinza_Dx: DINT;
*)	
	Pwr_status_C1: BOOL;
	Pwr_status_C2: BOOL;
	Pwr_status_C3: BOOL;
	Pwr_status_C4: BOOL;
	Pwr_Status_Larg_Bracci: BOOL;
	Pwr_Status_Pinza_Sx: BOOL;
	Pwr_Status_Pinza_Dx: BOOL;
	
	Pwr_Status_PTO_0: BOOL;
	Pwr_Status_PTO_1: BOOL;
	
	Tst_Home_Carrelli: BOOL;
	Tst_Home_Pinze: BOOL;

	Tts_Pos_Carrelli: BOOL;
	Tst_Pos_Pinze: BOOL;

	c1_pos_eseguito: BOOL;
	c2_pos_eseguito: BOOL;
	c3_pos_eseguito: BOOL;
	c4_pos_eseguito: BOOL;
	Larg_Bracci_pos_eseguito: BOOL;
	Pinza_Sx_pos_eseguito: BOOL;
	Pinza_Dx_pos_eseguito: BOOL;

	Tst_Corr_Carrello1: BOOL;
	Tst_Corr_Carrello2: BOOL;
	Tst_Corr_Carrello3: BOOL;
	Tst_Corr_Carrello4: BOOL;
	Tst_Corr_Larg_Bracci: BOOL;
	Tst_Corr_Pinza_Sx: BOOL;
	Tst_Corr_Pinza_Dx: BOOL;
	Tst_Corr_Centr1: BOOL;
	Tst_Corr_Centr2: BOOL;

	Acq_Carr: BOOL;
	Acq_Larg_Bracci_Colon: BOOL;
	Acq_Centr: BOOL;

	Unita_10X:BOOL;
	DI_Unita_10X:BOOL;
	
	Y_sblocco_Carrelli: BOOL;
	Y_sblocco_Pinze: BOOL;
	Y_sblocco_Larg_Bracci: BOOL;
	

	Done_SetPosition_C1: BOOL;
	Done_SetPosition_C2: BOOL;
	Done_SetPosition_C3: BOOL;
	Done_SetPosition_C4: BOOL;
	Done_SetPosition_Larg_Bracci: BOOL;
	Done_SetPosition_Pinza_Sx: BOOL;
	Done_SetPosition_Pinza_Dx: BOOL;
	DoneMoreRel_PTO_1: BOOL;
	
	Stato_Drv_Centr_1: BOOL;  //Steppers Ingresso Driver OK
	Stato_Drv_Centr_2: BOOL;  //Steppers Ingresso Driver OK
	
	Abil_Uscita_Centr_1: BOOL;
	Abil_Uscita_Centr_2: BOOL;
	
	Potenza_Attiva: BOOL;
	
	UM_Abil_Vol: BOOL;
	Abil_Power_Centr: BOOL;

	Centr1_Pag_Auto: BOOL;
	Centr2_Pag_Auto: BOOL;
	Centr1_Jog_Auto: BOOL;
	Centr2_Jog_Auto: BOOL;
	Pag_auto_riv: BOOL;
	
	Tst_Pos_Larg_Bracci:BOOL;
(*
	Actual_Position_Carrello_1: DINT;
	Actual_Position_Carrello_2: DINT;
	Actual_Position_Carrello_3: DINT;
	Actual_Position_Carrello_4: DINT;
	Actual_Position_Larg_Bracci: 	DINT;
	Actual_Position_Pinza_Sx: DINT;
	Actual_Position_Pinza_Dx: DINT;

	Actual_Position_Centratore_1: DINT;
	Actual_Position_Centratore_2: DINT;

//	Actual_Position_Volantino: 	INT;
*)
	Flag_SPos_Master_C1: BOOL;
	Flag_SPos_Master_C2: BOOL;
	Flag_SPos_Master_C3: BOOL;
	Flag_SPos_Master_C4: BOOL;
	Flag_SPos_Master_Bracci: BOOL;
	Flag_SPos_Master_Pinza_Sx: BOOL;
	Flag_SPos_Master_Pinza_Dx: BOOL;
	
	Flag_SPos_Slave_C1: BOOL;
	Flag_SPos_Slave_C2: BOOL;
	Flag_SPos_Slave_C3: BOOL;
	Flag_SPos_Slave_C4: BOOL;
	Flag_SPos_Slave_Bracci: BOOL;
	Flag_SPos_Slave_Pinza_Sx: BOOL;
	Flag_SPos_Slave_Pinza_Dx: BOOL;
	
	
//	Position_setting: BOOL;
	Larg_Bracci_setpos_eseguito: BOOL;
//	Pinxa_Sx_attivo: BOOL;
	Pinza_Sx_attivo: 	BOOL;
	Pinza_Sx_setpos_eseguito: BOOL;
	Pinza_Dx_attivo: 	BOOL;
//	Pinxa_Dx_attivo: BOOL;
	Pinza_Dx_setpos_eseguito: BOOL;
//	Token: BOOL;
//	Reverse_Token: BOOL;
//	Cancella_allarmi: BOOL;
	C1_setpos_eseguito: BOOL;
	C2_setpos_eseguito: BOOL;
	C3_setpos_eseguito: BOOL;
	C4_setpos_eseguito: BOOL;
	
	Direction_ILS: DINT;

	TargetPos_1: DWORD;
END_VAR

// MyController/Application/Global_VAR/GVL_HMI
VAR_GLOBAL
	Alm_Quota_Min_C1_C3: BOOL;
	Alm_Quota_Max_C1_C3: BOOL;
	Alm_Quota_Min_C2_C4: BOOL;
	Alm_Quota_Max_C2_C4: BOOL;
	Alm_Quota_Min_Larg_Bracci: BOOL;
	Alm_Quota_Max_Larg_Bracci: BOOL;
	Alm_Quota_Min_Pinze: BOOL;
	Alm_Quota_Max_Pinze: BOOL;
	
	Vis_Enc_Volantino: DINT;
	
	
END_VAR

// MyController/Application/Global_VAR/GVL_IO
VAR_GLOBAL
END_VAR

// MyController/Application/Global_VAR/PersistentVars
VAR_GLOBAL PERSISTENT RETAIN
	
Sviluppo_encodervol: INT;
Div_encoder: INT;


//Referenziato Pers.
Ref_Carrello_1: BOOL;
Ref_Carrello_2: BOOL;
Ref_Carrello_3: BOOL;
Ref_Carrello_4: BOOL;
Ref_Larg_Bracci: BOOL;
Ref_Pinza_Sx: BOOL;
Ref_Pinza_Dx: BOOL;
Centr1_home_noto: BOOL;
Centr2_home_noto: BOOL;

//in posizione
In_Pos_Carrello_1: BOOL;
In_Pos_Carrello_2: BOOL;
In_Pos_Carrello_3: BOOL;
In_Pos_Carrello_4: BOOL;
In_Pos_Larg_Bracci: BOOL;
In_Pos_Pinza_Sx: BOOL;
In_Pos_Pinza_Dx: BOOL;

//Backup Posizione (INSERISCI CONDIZIONI CHE ATTIVANO SET)

Position_Carrello_1: DINT;
Position_Carrello_2: DINT;
Position_Carrello_3: DINT;
Position_Carrello_4: DINT;
Position_Larg_Bracci: DINT;
Position_Pinza_Sx: DINT;
Position_Pinza_Dx: DINT;

END_VAR

// MyController/Application/Global_VAR/GVL_Motion
VAR_GLOBAL
	FB_ILS_Carrello_1: FB_ILS;
	FB_ILS_Carrello_2: FB_ILS;
	FB_ILS_Carrello_3: FB_ILS;
	FB_ILS_Carrello_4: FB_ILS;
	FB_ILS_Larg_Bracci: FB_ILS;
	FB_ILS_Pinza_Sx: FB_ILS;
	FB_ILS_Pinza_Dx: FB_ILS;
	
	FB_Stepper_Centratore_1: FB_Steppers;
	FB_Steppers_Centratore_2: FB_Steppers;
	
	Kt_carrelli: INT;
	Kt_larg_bracci: INT;
	Kt_pinze: INT;
	Kt_centratori: INT;
	q_error_absolute: BOOL;
END_VAR

// MyController/Application/P0_Main
PROGRAM P0_Main
VAR
	
END_VAR

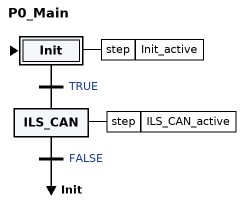
INITIAL_STEP Init:
    Init_active(N);  // step action
END_STEP
TRANSITION FROM Init TO ILS_CAN
    := TRUE;
END_TRANSITION
STEP ILS_CAN:
    ILS_CAN_active(N);  // step action
END_STEP
TRANSITION FROM ILS_CAN TO Init
    := FALSE;
END_TRANSITION

ACTION Init_active:
//Inizializzazione formati limite - dmm	
	M241_Largh_Max_Scat:= 4200; //C1-C3
	M241_Largh_Min_Scat:= 240; //C1-C3
	M241_Lungh_Max_Scat:= 6100; //C2-C4
	M241_Lungh_Min_Scat:= 480; //C2-C4 
	
//inizializzazione rapporti di trasmissione regolazioni
Kt_carrelli:= 1800;			//20000 * 3.6 / 4 impulsi per mm di avanzamento
Kt_Larg_Bracci:= 480;		//20000 * 1.92 / 8 impulsi per mm di avanzamento
Kt_Pinze:= 2000;		//20000 * 2 / 6 impulsi per mm di avanzamento - da dividere per 3 nei calcoli successivi

//Abilitazione iniziale contatore encoder volantino
Enc_Vol_Restart:= TRUE;

//Inizializzazione Volantino - MoveAdd 
Vel_Add_Carrello_1:= Kt_carrelli / 4;
Vel_Add_Carrello_2:= Kt_carrelli / 4;
Vel_Add_Carrello_3:= Kt_carrelli / 4;
Vel_Add_Carrello_4:= Kt_carrelli / 4;
Vel_Add_Larg_Bracci:= Kt_Larg_Bracci / 2;
Vel_Add_Pinza_Sx:= Kt_Pinze / 6;
Vel_Add_Pinza_Dx:= Kt_Pinze / 6;

//Inizializzazione Homing Mode 
HomingMode_Carrello_1:= 3;
VHome_Carrello_1:= Kt_carrelli / 4;
VoutHome_Carrello_1:= Kt_carrelli / 4;
HomingMode_Carrello_2:= 3;
VHome_Carrello_2:= Kt_carrelli / 4;
VoutHome_Carrello_2:= Kt_carrelli / 4;
HomingMode_Carrello_3:= 3;
VHome_Carrello_3:= Kt_carrelli / 4;
VoutHome_Carrello_3:= Kt_carrelli / 4;
HomingMode_Carrello_4:= 3;
VHome_Carrello_4:= Kt_carrelli / 4;
VoutHome_Carrello_4:= Kt_carrelli / 4;

HomingMode_Larg_Bracci:= 3;
VHome_Larg_Bracci:= Kt_Larg_Bracci / 2;
VoutHome_Larg_Bracci:= Kt_Larg_Bracci / 2;
HomingMode_Pinza_Sx:= 3;
VHome_Pinza_Sx:= Kt_Pinze / 6;
VoutHome_Pinza_Sx:= Kt_Pinze / 6;
HomingMode_Pinza_Dx:= 3;
VHome_Pinza_Dx:= Kt_Pinze / 6;
VoutHome_Pinza_Dx:= Kt_Pinze / 6;

PoutHome_Carrello_1:= 5000000;
PDisHome_Carrello_1:= 2000;
PoutHome_Carrello_2:= 5000000;
PDisHome_Carrello_2:= 2000;
PoutHome_Carrello_3:= 5000000;
PDisHome_Carrello_3:= 2000;
PoutHome_Carrello_4:= 5000000;
PDisHome_Carrello_4:= 2000;
PoutHome_Pinza_Sx:= 10000000;
PDisHome_Pinza_Sx:= 2000;
PoutHome_Pinza_Dx:= 10000000;
PDisHome_Pinza_Dx:= 2000;
PoutHome_Larg_Bracci:= 4000000;
PDisHome_Larg_Bracci:= 2000;

//Tip Jog
Tip_Jog_Carrello_1:= 100;
Tip_Jog_Carrello_2:= 100;
Tip_Jog_Carrello_3:= 100;
Tip_Jog_Carrello_4:= 100;
Tip_Jog_Larg_Bracci:= 100;
Tip_Jog_Pinza_Sx:= 100; 
Tip_Jog_Pinza_Dx:= 100;

//Inizializzazione Positon Mode 
Vel_Abs_Carrello_1:= Kt_carrelli / 4;
Vel_Abs_Carrello_2:= Kt_carrelli / 4;
Vel_Abs_Carrello_3:= Kt_carrelli / 4;
Vel_Abs_Carrello_4:= Kt_carrelli / 4;
Vel_Abs_Larg_Bracci:= Kt_Larg_Bracci / 2;
Vel_Abs_Pinza_Sx:= Kt_Pinze / 6;
Vel_Abs_Pinza_Dx:= Kt_Pinze / 6;
END_ACTION

ACTION ILS_CAN_active:
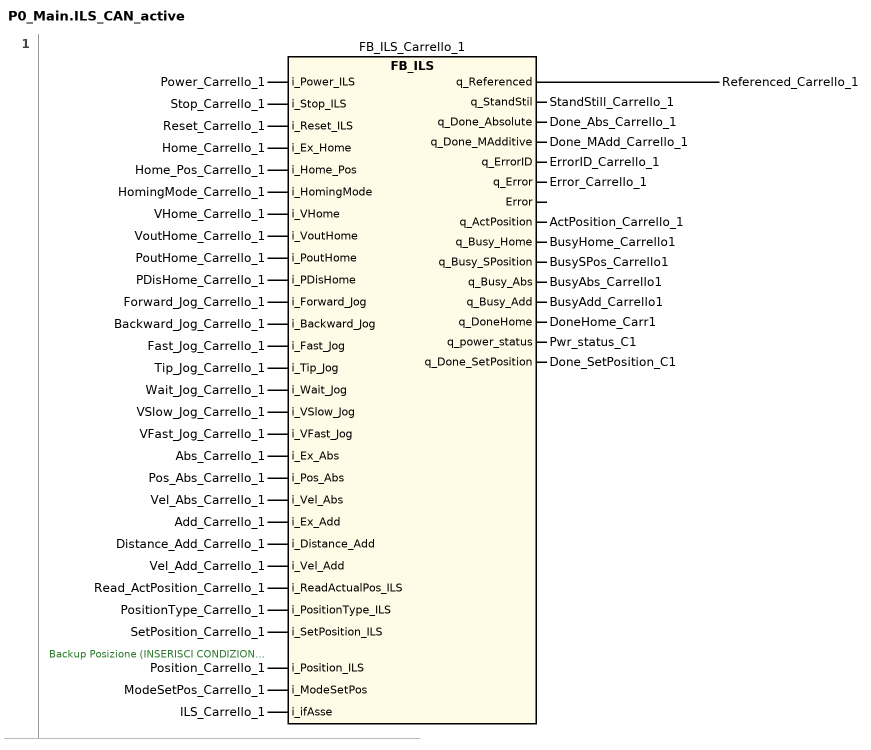
// NETWORK 1
//   Position_Carrello_1: Backup Posizione (INSERISCI CONDIZIONI CHE ATTIVANO SET)
FB_ILS_Carrello_1(
    i_Power_ILS := Power_Carrello_1,
    i_Stop_ILS := Stop_Carrello_1,
    i_Reset_ILS := Reset_Carrello_1,
    i_Ex_Home := Home_Carrello_1,
    i_Home_Pos := Home_Pos_Carrello_1,
    i_HomingMode := HomingMode_Carrello_1,
    i_VHome := VHome_Carrello_1,
    i_VoutHome := VoutHome_Carrello_1,
    i_PoutHome := PoutHome_Carrello_1,
    i_PDisHome := PDisHome_Carrello_1,
    i_Forward_Jog := Forward_Jog_Carrello_1,
    i_Backward_Jog := Backward_Jog_Carrello_1,
    i_Fast_Jog := Fast_Jog_Carrello_1,
    i_Tip_Jog := Tip_Jog_Carrello_1,
    i_Wait_Jog := Wait_Jog_Carrello_1,
    i_VSlow_Jog := VSlow_Jog_Carrello_1,
    i_VFast_Jog := VFast_Jog_Carrello_1,
    i_Ex_Abs := Abs_Carrello_1,
    i_Pos_Abs := Pos_Abs_Carrello_1,
    i_Vel_Abs := Vel_Abs_Carrello_1,
    i_Ex_Add := Add_Carrello_1,
    i_Distance_Add := Distance_Add_Carrello_1,
    i_Vel_Add := Vel_Add_Carrello_1,
    i_ReadActualPos_ILS := Read_ActPosition_Carrello_1,
    i_PositionType_ILS := PositionType_Carrello_1,
    i_SetPosition_ILS := SetPosition_Carrello_1,
    i_Position_ILS := Position_Carrello_1,
    i_ModeSetPos := ModeSetPos_Carrello_1,
    i_ifAsse := ILS_Carrello_1,
    q_StandStil => StandStill_Carrello_1,
    q_Done_Absolute => Done_Abs_Carrello_1,
    q_Done_MAdditive => Done_MAdd_Carrello_1,
    q_ErrorID => ErrorID_Carrello_1,
    q_Error => Error_Carrello_1,
    q_ActPosition => ActPosition_Carrello_1,
    q_Busy_Home => BusyHome_Carrello1,
    q_Busy_SPosition => BusySPos_Carrello1,
    q_Busy_Abs => BusyAbs_Carrello1,
    q_Busy_Add => BusyAdd_Carrello1,
    q_DoneHome => DoneHome_Carr1,
    q_power_status => Pwr_status_C1,
    q_Done_SetPosition => Done_SetPosition_C1); // FB_ILS
Referenced_Carrello_1 := FB_ILS_Carrello_1.q_Referenced;

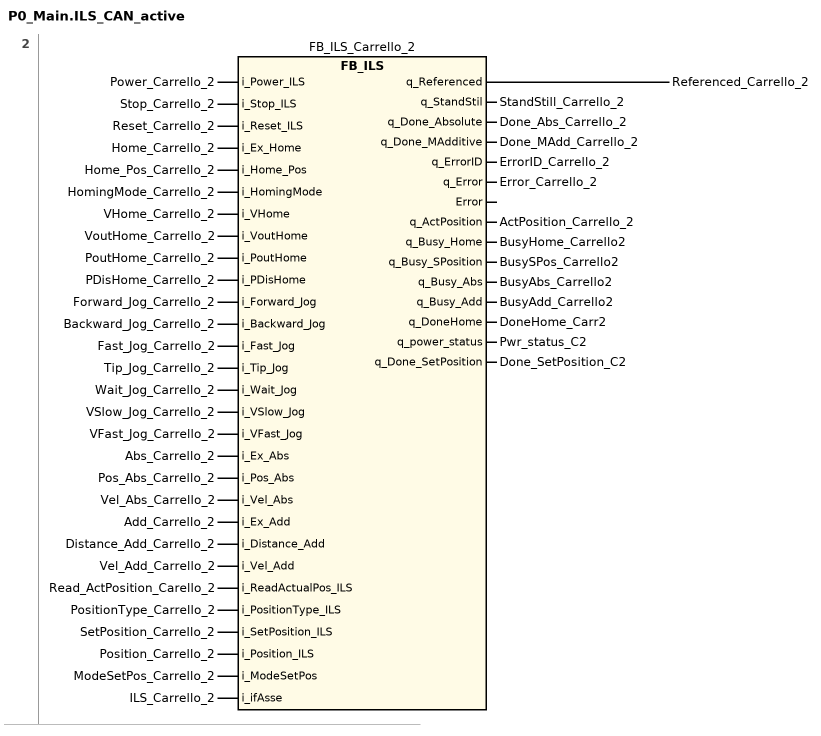
// NETWORK 2
FB_ILS_Carrello_2(
    i_Power_ILS := Power_Carrello_2,
    i_Stop_ILS := Stop_Carrello_2,
    i_Reset_ILS := Reset_Carrello_2,
    i_Ex_Home := Home_Carrello_2,
    i_Home_Pos := Home_Pos_Carrello_2,
    i_HomingMode := HomingMode_Carrello_2,
    i_VHome := VHome_Carrello_2,
    i_VoutHome := VoutHome_Carrello_2,
    i_PoutHome := PoutHome_Carrello_2,
    i_PDisHome := PDisHome_Carrello_2,
    i_Forward_Jog := Forward_Jog_Carrello_2,
    i_Backward_Jog := Backward_Jog_Carrello_2,
    i_Fast_Jog := Fast_Jog_Carrello_2,
    i_Tip_Jog := Tip_Jog_Carrello_2,
    i_Wait_Jog := Wait_Jog_Carrello_2,
    i_VSlow_Jog := VSlow_Jog_Carrello_2,
    i_VFast_Jog := VFast_Jog_Carrello_2,
    i_Ex_Abs := Abs_Carrello_2,
    i_Pos_Abs := Pos_Abs_Carrello_2,
    i_Vel_Abs := Vel_Abs_Carrello_2,
    i_Ex_Add := Add_Carrello_2,
    i_Distance_Add := Distance_Add_Carrello_2,
    i_Vel_Add := Vel_Add_Carrello_2,
    i_ReadActualPos_ILS := Read_ActPosition_Carello_2,
    i_PositionType_ILS := PositionType_Carrello_2,
    i_SetPosition_ILS := SetPosition_Carrello_2,
    i_Position_ILS := Position_Carrello_2,
    i_ModeSetPos := ModeSetPos_Carrello_2,
    i_ifAsse := ILS_Carrello_2,
    q_StandStil => StandStill_Carrello_2,
    q_Done_Absolute => Done_Abs_Carrello_2,
    q_Done_MAdditive => Done_MAdd_Carrello_2,
    q_ErrorID => ErrorID_Carrello_2,
    q_Error => Error_Carrello_2,
    q_ActPosition => ActPosition_Carrello_2,
    q_Busy_Home => BusyHome_Carrello2,
    q_Busy_SPosition => BusySPos_Carrello2,
    q_Busy_Abs => BusyAbs_Carrello2,
    q_Busy_Add => BusyAdd_Carrello2,
    q_DoneHome => DoneHome_Carr2,
    q_power_status => Pwr_status_C2,
    q_Done_SetPosition => Done_SetPosition_C2); // FB_ILS
Referenced_Carrello_2 := FB_ILS_Carrello_2.q_Referenced;

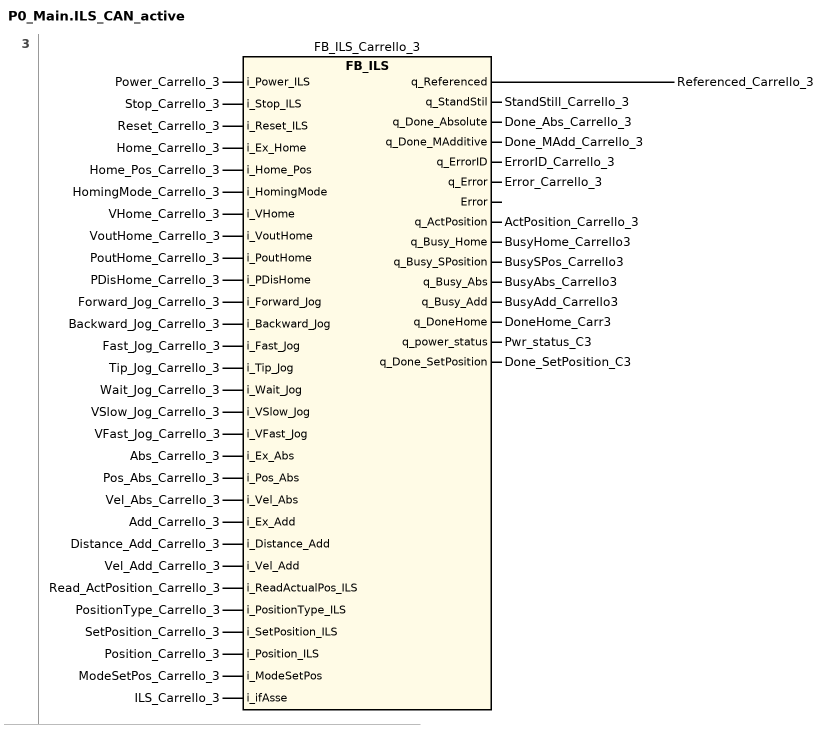
// NETWORK 3
FB_ILS_Carrello_3(
    i_Power_ILS := Power_Carrello_3,
    i_Stop_ILS := Stop_Carrello_3,
    i_Reset_ILS := Reset_Carrello_3,
    i_Ex_Home := Home_Carrello_3,
    i_Home_Pos := Home_Pos_Carrello_3,
    i_HomingMode := HomingMode_Carrello_3,
    i_VHome := VHome_Carrello_3,
    i_VoutHome := VoutHome_Carrello_3,
    i_PoutHome := PoutHome_Carrello_3,
    i_PDisHome := PDisHome_Carrello_3,
    i_Forward_Jog := Forward_Jog_Carrello_3,
    i_Backward_Jog := Backward_Jog_Carrello_3,
    i_Fast_Jog := Fast_Jog_Carrello_3,
    i_Tip_Jog := Tip_Jog_Carrello_3,
    i_Wait_Jog := Wait_Jog_Carrello_3,
    i_VSlow_Jog := VSlow_Jog_Carrello_3,
    i_VFast_Jog := VFast_Jog_Carrello_3,
    i_Ex_Abs := Abs_Carrello_3,
    i_Pos_Abs := Pos_Abs_Carrello_3,
    i_Vel_Abs := Vel_Abs_Carrello_3,
    i_Ex_Add := Add_Carrello_3,
    i_Distance_Add := Distance_Add_Carrello_3,
    i_Vel_Add := Vel_Add_Carrello_3,
    i_ReadActualPos_ILS := Read_ActPosition_Carrello_3,
    i_PositionType_ILS := PositionType_Carrello_3,
    i_SetPosition_ILS := SetPosition_Carrello_3,
    i_Position_ILS := Position_Carrello_3,
    i_ModeSetPos := ModeSetPos_Carrello_3,
    i_ifAsse := ILS_Carrello_3,
    q_StandStil => StandStill_Carrello_3,
    q_Done_Absolute => Done_Abs_Carrello_3,
    q_Done_MAdditive => Done_MAdd_Carrello_3,
    q_ErrorID => ErrorID_Carrello_3,
    q_Error => Error_Carrello_3,
    q_ActPosition => ActPosition_Carrello_3,
    q_Busy_Home => BusyHome_Carrello3,
    q_Busy_SPosition => BusySPos_Carrello3,
    q_Busy_Abs => BusyAbs_Carrello3,
    q_Busy_Add => BusyAdd_Carrello3,
    q_DoneHome => DoneHome_Carr3,
    q_power_status => Pwr_status_C3,
    q_Done_SetPosition => Done_SetPosition_C3); // FB_ILS
Referenced_Carrello_3 := FB_ILS_Carrello_3.q_Referenced;

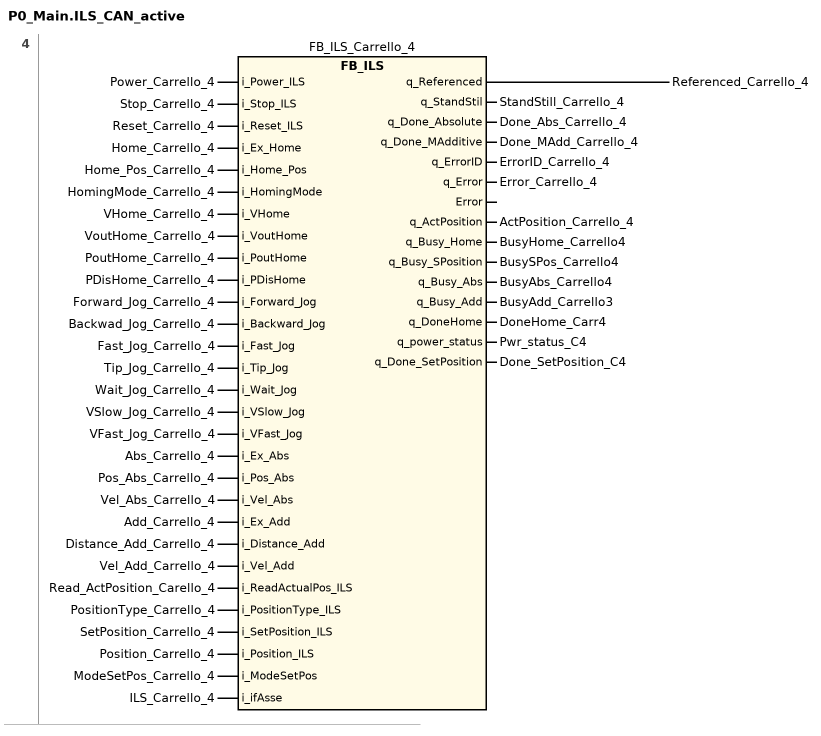
// NETWORK 4
FB_ILS_Carrello_4(
    i_Power_ILS := Power_Carrello_4,
    i_Stop_ILS := Stop_Carrello_4,
    i_Reset_ILS := Reset_Carrello_4,
    i_Ex_Home := Home_Carrello_4,
    i_Home_Pos := Home_Pos_Carrello_4,
    i_HomingMode := HomingMode_Carrello_4,
    i_VHome := VHome_Carrello_4,
    i_VoutHome := VoutHome_Carrello_4,
    i_PoutHome := PoutHome_Carrello_4,
    i_PDisHome := PDisHome_Carrello_4,
    i_Forward_Jog := Forward_Jog_Carrello_4,
    i_Backward_Jog := Backwad_Jog_Carrello_4,
    i_Fast_Jog := Fast_Jog_Carrello_4,
    i_Tip_Jog := Tip_Jog_Carrello_4,
    i_Wait_Jog := Wait_Jog_Carrello_4,
    i_VSlow_Jog := VSlow_Jog_Carrello_4,
    i_VFast_Jog := VFast_Jog_Carrello_4,
    i_Ex_Abs := Abs_Carrello_4,
    i_Pos_Abs := Pos_Abs_Carrello_4,
    i_Vel_Abs := Vel_Abs_Carrello_4,
    i_Ex_Add := Add_Carrello_4,
    i_Distance_Add := Distance_Add_Carrello_4,
    i_Vel_Add := Vel_Add_Carrello_4,
    i_ReadActualPos_ILS := Read_ActPosition_Carello_4,
    i_PositionType_ILS := PositionType_Carrello_4,
    i_SetPosition_ILS := SetPosition_Carrello_4,
    i_Position_ILS := Position_Carrello_4,
    i_ModeSetPos := ModeSetPos_Carrello_4,
    i_ifAsse := ILS_Carrello_4,
    q_StandStil => StandStill_Carrello_4,
    q_Done_Absolute => Done_Abs_Carrello_4,
    q_Done_MAdditive => Done_MAdd_Carrello_4,
    q_ErrorID => ErrorID_Carrello_4,
    q_Error => Error_Carrello_4,
    q_ActPosition => ActPosition_Carrello_4,
    q_Busy_Home => BusyHome_Carrello4,
    q_Busy_SPosition => BusySPos_Carrello4,
    q_Busy_Abs => BusyAbs_Carrello4,
    q_Busy_Add => BusyAdd_Carrello3,
    q_DoneHome => DoneHome_Carr4,
    q_power_status => Pwr_status_C4,
    q_Done_SetPosition => Done_SetPosition_C4); // FB_ILS
Referenced_Carrello_4 := FB_ILS_Carrello_4.q_Referenced;

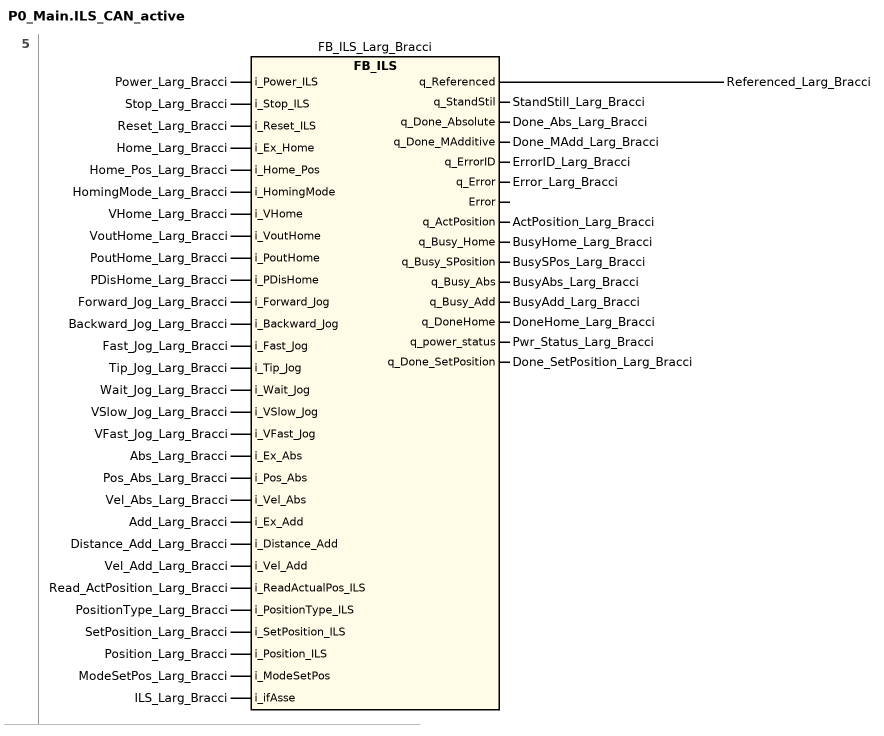
// NETWORK 5
FB_ILS_Larg_Bracci(
    i_Power_ILS := Power_Larg_Bracci,
    i_Stop_ILS := Stop_Larg_Bracci,
    i_Reset_ILS := Reset_Larg_Bracci,
    i_Ex_Home := Home_Larg_Bracci,
    i_Home_Pos := Home_Pos_Larg_Bracci,
    i_HomingMode := HomingMode_Larg_Bracci,
    i_VHome := VHome_Larg_Bracci,
    i_VoutHome := VoutHome_Larg_Bracci,
    i_PoutHome := PoutHome_Larg_Bracci,
    i_PDisHome := PDisHome_Larg_Bracci,
    i_Forward_Jog := Forward_Jog_Larg_Bracci,
    i_Backward_Jog := Backward_Jog_Larg_Bracci,
    i_Fast_Jog := Fast_Jog_Larg_Bracci,
    i_Tip_Jog := Tip_Jog_Larg_Bracci,
    i_Wait_Jog := Wait_Jog_Larg_Bracci,
    i_VSlow_Jog := VSlow_Jog_Larg_Bracci,
    i_VFast_Jog := VFast_Jog_Larg_Bracci,
    i_Ex_Abs := Abs_Larg_Bracci,
    i_Pos_Abs := Pos_Abs_Larg_Bracci,
    i_Vel_Abs := Vel_Abs_Larg_Bracci,
    i_Ex_Add := Add_Larg_Bracci,
    i_Distance_Add := Distance_Add_Larg_Bracci,
    i_Vel_Add := Vel_Add_Larg_Bracci,
    i_ReadActualPos_ILS := Read_ActPosition_Larg_Bracci,
    i_PositionType_ILS := PositionType_Larg_Bracci,
    i_SetPosition_ILS := SetPosition_Larg_Bracci,
    i_Position_ILS := Position_Larg_Bracci,
    i_ModeSetPos := ModeSetPos_Larg_Bracci,
    i_ifAsse := ILS_Larg_Bracci,
    q_StandStil => StandStill_Larg_Bracci,
    q_Done_Absolute => Done_Abs_Larg_Bracci,
    q_Done_MAdditive => Done_MAdd_Larg_Bracci,
    q_ErrorID => ErrorID_Larg_Bracci,
    q_Error => Error_Larg_Bracci,
    q_ActPosition => ActPosition_Larg_Bracci,
    q_Busy_Home => BusyHome_Larg_Bracci,
    q_Busy_SPosition => BusySPos_Larg_Bracci,
    q_Busy_Abs => BusyAbs_Larg_Bracci,
    q_Busy_Add => BusyAdd_Larg_Bracci,
    q_DoneHome => DoneHome_Larg_Bracci,
    q_power_status => Pwr_Status_Larg_Bracci,
    q_Done_SetPosition => Done_SetPosition_Larg_Bracci); // FB_ILS
Referenced_Larg_Bracci := FB_ILS_Larg_Bracci.q_Referenced;

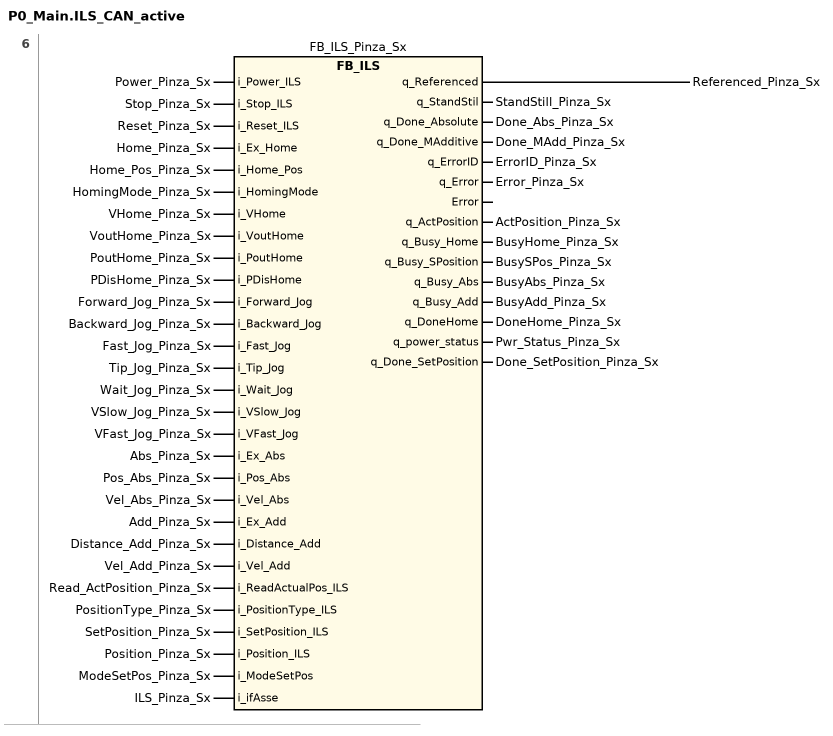
// NETWORK 6
FB_ILS_Pinza_Sx(
    i_Power_ILS := Power_Pinza_Sx,
    i_Stop_ILS := Stop_Pinza_Sx,
    i_Reset_ILS := Reset_Pinza_Sx,
    i_Ex_Home := Home_Pinza_Sx,
    i_Home_Pos := Home_Pos_Pinza_Sx,
    i_HomingMode := HomingMode_Pinza_Sx,
    i_VHome := VHome_Pinza_Sx,
    i_VoutHome := VoutHome_Pinza_Sx,
    i_PoutHome := PoutHome_Pinza_Sx,
    i_PDisHome := PDisHome_Pinza_Sx,
    i_Forward_Jog := Forward_Jog_Pinza_Sx,
    i_Backward_Jog := Backward_Jog_Pinza_Sx,
    i_Fast_Jog := Fast_Jog_Pinza_Sx,
    i_Tip_Jog := Tip_Jog_Pinza_Sx,
    i_Wait_Jog := Wait_Jog_Pinza_Sx,
    i_VSlow_Jog := VSlow_Jog_Pinza_Sx,
    i_VFast_Jog := VFast_Jog_Pinza_Sx,
    i_Ex_Abs := Abs_Pinza_Sx,
    i_Pos_Abs := Pos_Abs_Pinza_Sx,
    i_Vel_Abs := Vel_Abs_Pinza_Sx,
    i_Ex_Add := Add_Pinza_Sx,
    i_Distance_Add := Distance_Add_Pinza_Sx,
    i_Vel_Add := Vel_Add_Pinza_Sx,
    i_ReadActualPos_ILS := Read_ActPosition_Pinza_Sx,
    i_PositionType_ILS := PositionType_Pinza_Sx,
    i_SetPosition_ILS := SetPosition_Pinza_Sx,
    i_Position_ILS := Position_Pinza_Sx,
    i_ModeSetPos := ModeSetPos_Pinza_Sx,
    i_ifAsse := ILS_Pinza_Sx,
    q_StandStil => StandStill_Pinza_Sx,
    q_Done_Absolute => Done_Abs_Pinza_Sx,
    q_Done_MAdditive => Done_MAdd_Pinza_Sx,
    q_ErrorID => ErrorID_Pinza_Sx,
    q_Error => Error_Pinza_Sx,
    q_ActPosition => ActPosition_Pinza_Sx,
    q_Busy_Home => BusyHome_Pinza_Sx,
    q_Busy_SPosition => BusySPos_Pinza_Sx,
    q_Busy_Abs => BusyAbs_Pinza_Sx,
    q_Busy_Add => BusyAdd_Pinza_Sx,
    q_DoneHome => DoneHome_Pinza_Sx,
    q_power_status => Pwr_Status_Pinza_Sx,
    q_Done_SetPosition => Done_SetPosition_Pinza_Sx); // FB_ILS
Referenced_Pinza_Sx := FB_ILS_Pinza_Sx.q_Referenced;

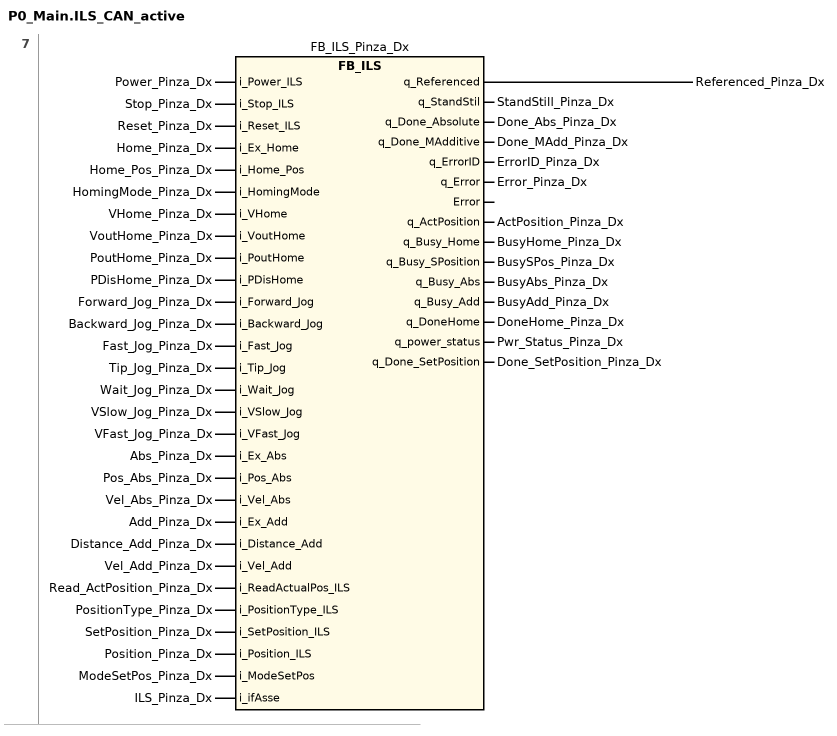
// NETWORK 7
FB_ILS_Pinza_Dx(
    i_Power_ILS := Power_Pinza_Dx,
    i_Stop_ILS := Stop_Pinza_Dx,
    i_Reset_ILS := Reset_Pinza_Dx,
    i_Ex_Home := Home_Pinza_Dx,
    i_Home_Pos := Home_Pos_Pinza_Dx,
    i_HomingMode := HomingMode_Pinza_Dx,
    i_VHome := VHome_Pinza_Dx,
    i_VoutHome := VoutHome_Pinza_Dx,
    i_PoutHome := PoutHome_Pinza_Dx,
    i_PDisHome := PDisHome_Pinza_Dx,
    i_Forward_Jog := Forward_Jog_Pinza_Dx,
    i_Backward_Jog := Backward_Jog_Pinza_Dx,
    i_Fast_Jog := Fast_Jog_Pinza_Dx,
    i_Tip_Jog := Tip_Jog_Pinza_Dx,
    i_Wait_Jog := Wait_Jog_Pinza_Dx,
    i_VSlow_Jog := VSlow_Jog_Pinza_Dx,
    i_VFast_Jog := VFast_Jog_Pinza_Dx,
    i_Ex_Abs := Abs_Pinza_Dx,
    i_Pos_Abs := Pos_Abs_Pinza_Dx,
    i_Vel_Abs := Vel_Abs_Pinza_Dx,
    i_Ex_Add := Add_Pinza_Dx,
    i_Distance_Add := Distance_Add_Pinza_Dx,
    i_Vel_Add := Vel_Add_Pinza_Dx,
    i_ReadActualPos_ILS := Read_ActPosition_Pinza_Dx,
    i_PositionType_ILS := PositionType_Pinza_Dx,
    i_SetPosition_ILS := SetPosition_Pinza_Dx,
    i_Position_ILS := Position_Pinza_Dx,
    i_ModeSetPos := ModeSetPos_Pinza_Dx,
    i_ifAsse := ILS_Pinza_Dx,
    q_StandStil => StandStill_Pinza_Dx,
    q_Done_Absolute => Done_Abs_Pinza_Dx,
    q_Done_MAdditive => Done_MAdd_Pinza_Dx,
    q_ErrorID => ErrorID_Pinza_Dx,
    q_Error => Error_Pinza_Dx,
    q_ActPosition => ActPosition_Pinza_Dx,
    q_Busy_Home => BusyHome_Pinza_Dx,
    q_Busy_SPosition => BusySPos_Pinza_Dx,
    q_Busy_Abs => BusyAbs_Pinza_Dx,
    q_Busy_Add => BusyAdd_Pinza_Dx,
    q_DoneHome => DoneHome_Pinza_Dx,
    q_power_status => Pwr_Status_Pinza_Dx,
    q_Done_SetPosition => Done_SetPosition_Pinza_Dx); // FB_ILS
Referenced_Pinza_Dx := FB_ILS_Pinza_Dx.q_Referenced;
END_ACTION

END_PROGRAM

// MyController/Application/FB_ILS
FUNCTION_BLOCK FB_ILS
VAR_INPUT
	
	
	i_Power_ILS: BOOL;
	i_Stop_ILS: BOOL;
	i_Reset_ILS: BOOL;
	i_Ex_Home: BOOL;
	i_Home_Pos: DINT;
	i_HomingMode: UINT;
	i_VHome: UINT;
	i_VoutHome: UINT;
	i_PoutHome: DINT;
	i_PDisHome: DINT;
	i_Forward_Jog: BOOL;
	i_Backward_Jog: BOOL;
	i_Fast_Jog: BOOL;
	i_Tip_Jog: UINT;
	i_Wait_Jog: UINT;
	i_VSlow_Jog: INT;
	i_VFast_Jog: INT;
	i_Ex_Abs: BOOL;
	i_Pos_Abs: DINT;
	i_Vel_Abs: INT;
	i_Ex_Add: BOOL;
	i_Distance_Add: DINT;
	i_Vel_Add: INT;
	i_ReadActualPos_ILS: BOOL;
	i_PositionType_ILS: INT;
	i_SetPosition_ILS: BOOL;
	i_Position_ILS: DINT; 
	i_ModeSetPos: BOOL;
END_VAR
VAR_OUTPUT
	q_Referenced: BOOL;
	q_StandStil: BOOL;
	q_Done_Absolute: BOOL;
	q_Done_MAdditive: BOOL;
	q_ErrorID: WORD;
	q_Error: BOOL;
	Error: BOOL;
	q_ActPosition: DINT;
	q_Busy_Home: BOOL;
	q_Busy_SPosition: BOOL;
	q_Busy_Abs: BOOL;
	q_Busy_Add: BOOL;
	q_DoneHome: BOOL;
	q_power_status: BOOL;
	q_Done_SetPosition: BOOL;
END_VAR
VAR
	MC_Power_ILX_0: MC_Power_ILX;
	MC_Stop_ILX_0: MC_Stop_ILX;
	MC_Reset_ILX_0: MC_Reset_ILX;
	MC_Jog_ILX_0: MC_Jog_ILX;
	MC_ReadAxisError_ILX_0: MC_ReadAxisError_ILX;
	MC_ReadStatus_ILX_0: MC_ReadStatus_ILX;
	MC_Home_ILX_0: MC_Home_ILX;
	MC_MoveAbsolute_ILX_0: MC_MoveAbsolute_ILX;
	MC_MoveAdditive_ILX_0: MC_MoveAdditive_ILX;
	MC_ReadActualPosition_ILX_0: MC_ReadActualPosition_ILX;
	MC_SetPosition_ILX_0: MC_SetPosition_ILX;

	IO_write: BOOL;
	ConfigureIO_0: ConfigureIO_ILX;
	ConfigureIO_1: ConfigureIO_ILX;
	ConfigureIO_2: ConfigureIO_ILX;
	ConfigureIO_3: ConfigureIO_ILX;
	StoreParameters_ILX_0: SEM_ILX.StoreParameters_ILX;
	ILS_writeparametersdirection: SEM_ILX.MC_WriteParameter_ILX;
	Write_Dir: BOOL;
	Parameter_read: BOOL;
	Parameter_value_read: DINT;
	Prameter_read: MC_ReadParameter_ILX;
	I_O_read_ILX: MC_ReadDigitalInput_ILX;
	Input_value: BOOL;
	Number: INT;
	Par_number: UINT;
	Index: UINT;
	I_O_read: BOOL;
	Subindex: UINT;
END_VAR

VAR_IN_OUT
	i_ifAsse: Axis_Ref_ILX;
END_VAR

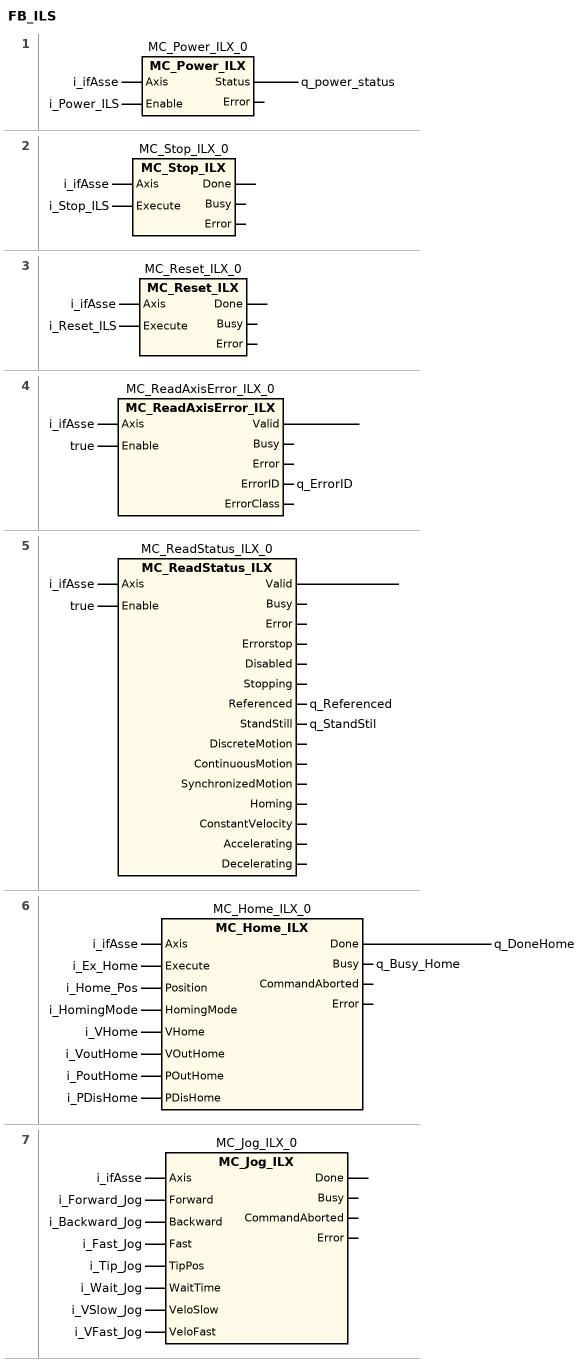
// NETWORK 1
MC_Power_ILX_0(Axis := i_ifAsse, Enable := i_Power_ILS); // MC_Power_ILX
q_power_status := MC_Power_ILX_0.Status;

// NETWORK 2
MC_Stop_ILX_0(Axis := i_ifAsse, Execute := i_Stop_ILS); // MC_Stop_ILX

// NETWORK 3
MC_Reset_ILX_0(Axis := i_ifAsse, Execute := i_Reset_ILS); // MC_Reset_ILX

// NETWORK 4
MC_ReadAxisError_ILX_0(Axis := i_ifAsse, Enable := true, ErrorID => q_ErrorID); // MC_ReadAxisError_ILX

// NETWORK 5
MC_ReadStatus_ILX_0(Axis := i_ifAsse, Enable := true, Referenced => q_Referenced, StandStill => q_StandStil); // MC_ReadStatus_ILX

// NETWORK 6
MC_Home_ILX_0(
    Axis := i_ifAsse,
    Execute := i_Ex_Home,
    Position := i_Home_Pos,
    HomingMode := i_HomingMode,
    VHome := i_VHome,
    VOutHome := i_VoutHome,
    POutHome := i_PoutHome,
    PDisHome := i_PDisHome,
    Busy => q_Busy_Home); // MC_Home_ILX
q_DoneHome := MC_Home_ILX_0.Done;

// NETWORK 7
MC_Jog_ILX_0(
    Axis := i_ifAsse,
    Forward := i_Forward_Jog,
    Backward := i_Backward_Jog,
    Fast := i_Fast_Jog,
    TipPos := i_Tip_Jog,
    WaitTime := i_Wait_Jog,
    VeloSlow := i_VSlow_Jog,
    VeloFast := i_VFast_Jog); // MC_Jog_ILX

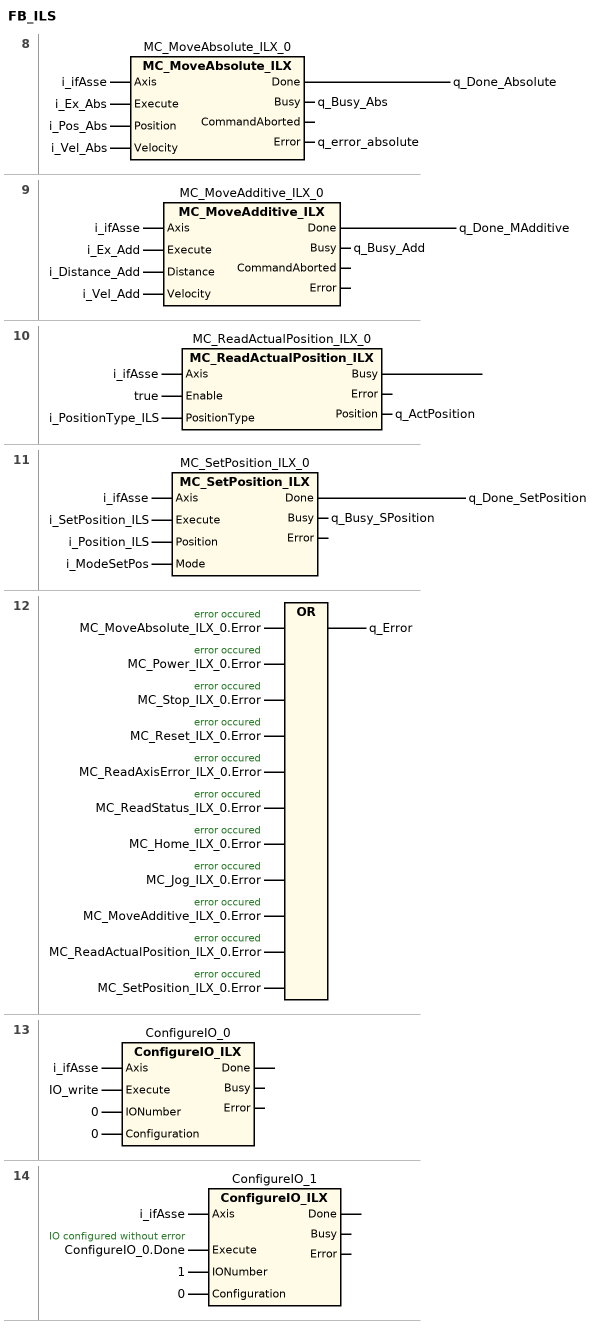
// NETWORK 8
MC_MoveAbsolute_ILX_0(
    Axis := i_ifAsse,
    Execute := i_Ex_Abs,
    Position := i_Pos_Abs,
    Velocity := i_Vel_Abs,
    Busy => q_Busy_Abs,
    Error => q_error_absolute); // MC_MoveAbsolute_ILX
q_Done_Absolute := MC_MoveAbsolute_ILX_0.Done;

// NETWORK 9
MC_MoveAdditive_ILX_0(
    Axis := i_ifAsse,
    Execute := i_Ex_Add,
    Distance := i_Distance_Add,
    Velocity := i_Vel_Add,
    Busy => q_Busy_Add); // MC_MoveAdditive_ILX
q_Done_MAdditive := MC_MoveAdditive_ILX_0.Done;

// NETWORK 10
MC_ReadActualPosition_ILX_0(
    Axis := i_ifAsse,
    Enable := true,
    PositionType := i_PositionType_ILS,
    Position => q_ActPosition); // MC_ReadActualPosition_ILX

// NETWORK 11
MC_SetPosition_ILX_0(
    Axis := i_ifAsse,
    Execute := i_SetPosition_ILS,
    Position := i_Position_ILS,
    Mode := i_ModeSetPos,
    Busy => q_Busy_SPosition); // MC_SetPosition_ILX
q_Done_SetPosition := MC_SetPosition_ILX_0.Done;

// NETWORK 12
//   MC_MoveAbsolute_ILX_0.Error: error occured
//   MC_Power_ILX_0.Error: error occured
//   MC_Stop_ILX_0.Error: error occured
//   MC_Reset_ILX_0.Error: error occured
//   MC_ReadAxisError_ILX_0.Error: error occured
//   MC_ReadStatus_ILX_0.Error: error occured
//   MC_Home_ILX_0.Error: error occured
//   MC_Jog_ILX_0.Error: error occured
//   MC_MoveAdditive_ILX_0.Error: error occured
//   MC_ReadActualPosition_ILX_0.Error: error occured
//   MC_SetPosition_ILX_0.Error: error occured
q_Error := MC_MoveAbsolute_ILX_0.Error OR MC_Power_ILX_0.Error OR MC_Stop_ILX_0.Error OR MC_Reset_ILX_0.Error OR MC_ReadAxisError_ILX_0.Error OR MC_ReadStatus_ILX_0.Error OR MC_Home_ILX_0.Error OR MC_Jog_ILX_0.Error OR MC_MoveAdditive_ILX_0.Error OR MC_ReadActualPosition_ILX_0.Error OR MC_SetPosition_ILX_0.Error;

// NETWORK 13
ConfigureIO_0(Axis := i_ifAsse, Execute := IO_write, IONumber := 0, Configuration := 0); // ConfigureIO_ILX

// NETWORK 14
//   ConfigureIO_0.Done: IO configured without error
ConfigureIO_1(Axis := i_ifAsse, Execute := ConfigureIO_0.Done, IONumber := 1, Configuration := 0); // ConfigureIO_ILX

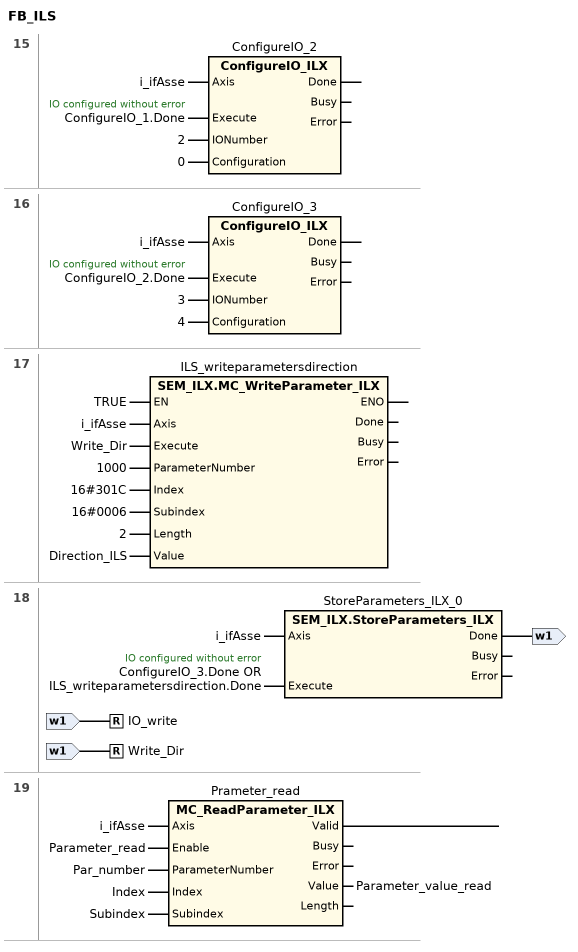
// NETWORK 15
//   ConfigureIO_1.Done: IO configured without error
ConfigureIO_2(Axis := i_ifAsse, Execute := ConfigureIO_1.Done, IONumber := 2, Configuration := 0); // ConfigureIO_ILX

// NETWORK 16
//   ConfigureIO_2.Done: IO configured without error
ConfigureIO_3(Axis := i_ifAsse, Execute := ConfigureIO_2.Done, IONumber := 3, Configuration := 4); // ConfigureIO_ILX

// NETWORK 17
ILS_writeparametersdirection(
    Axis := i_ifAsse,
    Execute := Write_Dir,
    ParameterNumber := 1000,
    Index := 16#301C,
    Subindex := 16#0006,
    Length := 2,
    Value := Direction_ILS); // SEM_ILX.MC_WriteParameter_ILX

// NETWORK 18
//   ConfigureIO_3.Done OR ILS_writeparametersdirection.Done: IO configured without error
StoreParameters_ILX_0(Axis := i_ifAsse, Execute := ConfigureIO_3.Done OR ILS_writeparametersdirection.Done); // SEM_ILX.StoreParameters_ILX
IO_write R= StoreParameters_ILX_0.Done;
Write_Dir R= StoreParameters_ILX_0.Done;

// NETWORK 19
Prameter_read(
    Axis := i_ifAsse,
    Enable := Parameter_read,
    ParameterNumber := Par_number,
    Index := Index,
    Subindex := Subindex,
    Value => Parameter_value_read); // MC_ReadParameter_ILX

END_FUNCTION_BLOCK

// MyController/Application/Programma/Clock_Encoder
PROGRAM  Clock_Encoder
VAR
	Blink_01s: BLINK;
	test: BOOL;
	
END_VAR

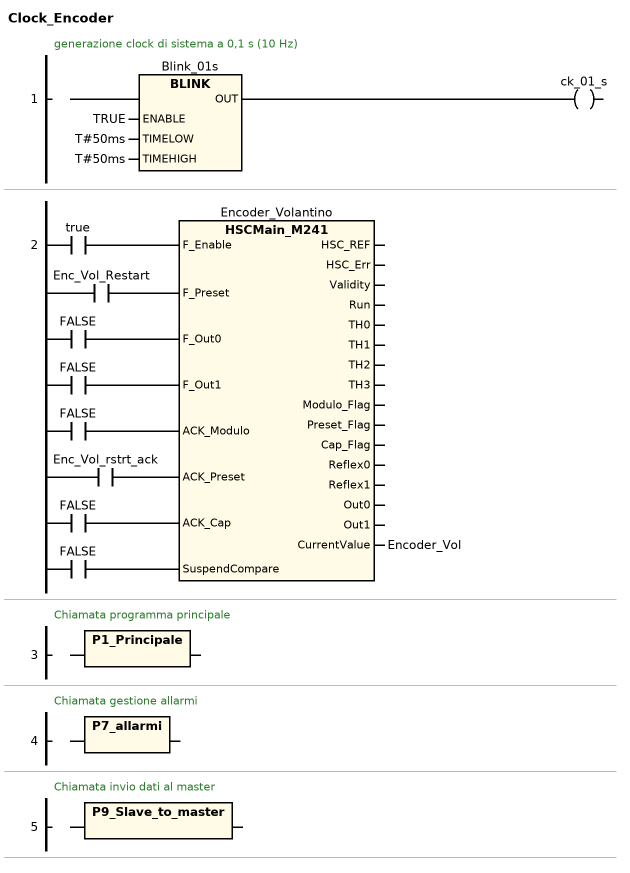
// NETWORK 1
// generazione clock di sistema a 0,1 s (10 Hz)
Blink_01s(ENABLE := TRUE, TIMELOW := T#50ms, TIMEHIGH := T#50ms); // BLINK
ck_01_s := Blink_01s.OUT;

// NETWORK 2
Encoder_Volantino(
    F_Enable := true,
    F_Preset := Enc_Vol_Restart,
    F_Out0 := FALSE,
    F_Out1 := FALSE,
    ACK_Modulo := FALSE,
    ACK_Preset := Enc_Vol_rstrt_ack,
    ACK_Cap := FALSE,
    SuspendCompare := FALSE,
    CurrentValue => Encoder_Vol); // HSCMain_M241

// NETWORK 3
// Chiamata programma principale
P1_Principale();

// NETWORK 4
// Chiamata gestione allarmi
P7_allarmi();

// NETWORK 5
// Chiamata invio dati al master
P9_Slave_to_master();

END_PROGRAM

// MyController/Application/Programma/P1_Principale
PROGRAM P1_Principale
VAR
	Start_Home_Gen: BOOL;
	Start_Pos_Gen: BOOL;
	R_Trig_Tst_Home_Carrelli: R_TRIG;
	R_Trig_Tst_Home_Larg_BracciColon: R_TRIG;
	R_Trig_Tst_Home_Centratori: R_TRIG;
	F_Tst_Home_Carrelli: F_TRIG;
	F_Tst_Home_Larg_BracciColon: F_TRIG;
	F_Tst_Home_Centratori: F_TRIG;
	
	R_clock01: R_TRIG;
	F_clock01: F_TRIG;
	C1_home_avviato: BOOL;
	T_stop_C1: TON;
	C1_pos_avviato: BOOL;
	T_avvio_corsa_C1: TON;
	
	C2_home_avviato: BOOL;
	T_stop_C2: TON;
	C2_pos_avviato: BOOL;
	T_avvio_corsa_C2: TON;
	
	C3_home_avviato: BOOL;
	T_stop_C3: TON;
	C3_pos_avviato: BOOL;
	T_avvio_corsa_C3: TON;
	
	C4_home_avviato: BOOL;
	T_stop_C4: TON;
	C4_pos_avviato: BOOL;
	T_avvio_corsa_C4: TON;
	
	Larg_Bracci_home_avviato: BOOL;
	T_stop_Larg_Bracci: TON;
	Larg_Bracci_pos_avviato: BOOL;
	T_avvio_corsa_Larg_Bracci: TON;
	
	Pinza_Sx_home_avviato: BOOL;
	T_stop_Pinza_Sx: TON;
	Pinza_Sx_pos_avviato: BOOL;
	T_avvio_corsa_Pinza_Sx: TON;
	
	Pinza_Dx_home_avviato: BOOL;
	T_stop_Pinza_Dx: TON;
	Pinza_Dx_pos_avviato: BOOL;
	T_avvio_corsa_Pinza_Dx: TON;
	
	Centr1_home_avviato: BOOL;
	T_stop_Centr1: TON;
	Centr1_pos_avviato: BOOL;
	T_avvio_corsa_Centr1: TON;
	
	Centr2_home_avviato: BOOL;
	T_stop_Centr2: TON;
	Centr2_pos_avviato: BOOL;
	T_avvio_corsa_Centr2: TON;
	
	T_exe_add_C1: TON;
	T_exe_add_C2: TON;
	T_exe_add_C3: TON;
	T_exe_add_C4: TON;
	T_exe_add_Larg_Bracci: TON;
	T_exe_add_Pinza_Sx: TON;
	T_exe_add_Pinza_Dx: TON;
	T_exe_add_centr1: TON;
	T_exe_add_centr2: TON;
	
	
	c1_home_eseguito: BOOL;
	c2_home_eseguito: BOOL;
	c3_home_eseguito: BOOL;
	c4_home_eseguito: BOOL;
	Larg_Bracci_home_eseguito: BOOL;
	Pinza_Sx_home_eseguito: BOOL;
	Pinza_Dx_home_eseguito: BOOL;
	centr1_home_eseguito: BOOL;
	centr2_home_eseguito: BOOL;
	centr1_pos_eseguito: BOOL;
	centr2_pos_eseguito: BOOL;

	C1_setpos_avviato: BOOL;
	C2_setpos_avviato: BOOL;
	C3_setpos_avviato: BOOL;
	C4_setpos_avviato: BOOL;
	F_C1_home: F_TRIG;
	F_C2_home: F_TRIG;
	F_C3_home: F_TRIG;
	F_C4_home: F_TRIG;
	F_C1_pos: F_TRIG;
	F_C2_pos: F_TRIG;
	F_C3_pos: F_TRIG;
	F_C4_pos: F_TRIG;
	da: INT;
	Pinza_Sx_setpos_avviato: BOOL;
	Pinza_Dx_setpos_avviato: BOOL;
	F_Larg_Bracci_Home: F_TRIG;
	F_Larg_Bracci_Pos: F_TRIG;
	F_Pinza_Sx_Home: F_TRIG;
	F_Pinza_Dx_Home: F_TRIG;
	F_Pinxa_Sx_Pos: F_TRIG;
	F_Pinxa_Dx_Pos: F_TRIG;
	Larg_Bracci_setpos_avviato: BOOL;
END_VAR

//Verifica reinizializzazione contatore
IF Enc_Vol_Restart THEN
	IF Encoder_Volantino.Preset_Flag THEN
		Enc_Vol_rstrt_ack:= TRUE;
	END_IF
	IF Encoder_Volantino.Validity THEN
		Enc_Vol_Restart:= FALSE;
		Last_Encoder_Vol:= 0;
	END_IF
ELSE 
	Enc_Vol_rstrt_ack:= FALSE;	
END_IF

// tempo di campionamento = 50 ms
R_clock01(CLK:= ck_01_s);
F_clock01(CLK:= ck_01_s);
sample_clock:= R_clock01.Q OR F_clock01.Q;

// gestione dello spostamento dell'encoder volantino
IF sample_clock THEN
	Delta_encvol:= Encoder_Vol - Last_Encoder_Vol;
	Last_Encoder_Vol:= Encoder_Vol;
END_IF

//comandi presenti assi regolazione 
//attivazione potenza
Power_Carrello_1:= (modo_regolazioni AND C1_enable OR Position_setting);
Power_Carrello_2:= (modo_regolazioni AND C2_enable OR Position_setting);
Power_Carrello_3:= (modo_regolazioni AND C3_enable OR Position_setting);
Power_Carrello_4:= (modo_regolazioni AND C4_enable OR Position_setting);
Power_Larg_Bracci:= (modo_regolazioni AND Larg_Bracci_enable OR Position_setting);
Power_Pinza_Sx:= (modo_regolazioni AND Pinza_Sx_enable OR Position_setting);
Power_Pinza_Dx:= (modo_regolazioni AND Pinza_Dx_enable OR Position_setting);

IF FB_ILS_Carrello_1.q_power_status AND (C1_home OR C1_position OR C1_jog OR C1_setpos) THEN
	C1_attivo:= TRUE;
ELSE
	C1_attivo:= FALSE;
END_IF

IF FB_ILS_Carrello_2.q_power_status AND (C2_home OR C2_position OR C2_jog OR C2_setpos) THEN
	C2_attivo:= TRUE;
ELSE
	C2_attivo:= FALSE;
END_IF

IF FB_ILS_Carrello_3.q_power_status AND (C3_home OR C3_position OR C3_jog OR C3_setpos) THEN
	C3_attivo:= TRUE;
ELSE
	C3_attivo:= FALSE;
END_IF

IF FB_ILS_Carrello_4.q_power_status AND (C4_home OR C4_position OR C4_jog OR C4_setpos) THEN
	C4_attivo:= TRUE;
ELSE
	C4_attivo:= FALSE;
END_IF

IF FB_ILS_Larg_Bracci.q_power_status AND (Larg_Bracci_home OR Larg_Bracci_position OR Larg_Bracci_jog OR Larg_Bracci_setpos) THEN
	Larg_Bracci_attivo:= TRUE;
ELSE
	Larg_Bracci_attivo:= FALSE;
END_IF

IF FB_ILS_Pinza_Sx.q_power_status AND (Pinza_Sx_home OR Pinza_Sx_position OR Pinza_Sx_jog OR Pinza_Sx_setpos) THEN
	Pinza_Sx_attivo:= TRUE;
ELSE
	Pinza_Sx_attivo:= FALSE;
END_IF

IF FB_ILS_Pinza_Dx.q_power_status AND (Pinza_Dx_home OR Pinza_Dx_position OR Pinza_Dx_jog OR Pinza_dx_setpos) THEN
	Pinza_Dx_attivo:= TRUE;
ELSE
	Pinza_Dx_attivo:= FALSE;
END_IF

//sblocco freno in presenza di attività dei relativi assi
IF sblocco_carrelli OR C1_attivo OR C2_attivo OR C3_attivo OR C4_attivo THEN
	Y_sblocco_Carrelli:= TRUE; 
ELSE
	Y_sblocco_Carrelli:=FALSE;
END_IF

IF sblocco_Pinze OR Larg_Bracci_attivo OR Pinza_Sx_attivo OR Pinza_Dx_attivo THEN
	Y_sblocco_Pinze:= TRUE; 
ELSE
	Y_sblocco_Pinze:=FALSE;
END_IF

//Scrittura Quote_Position (target di posizione secondo il comando da eseguire) 03.09.2018

IF NOT Alm_Quota_Max_C1_C3 AND NOT Alm_Quota_Min_C1_C3  THEN 
	Pos_Abs_Carrello_1:= Target_Pos_Carrello_1 * Kt_carrelli;
	Pos_Abs_Carrello_3:= Target_Pos_Carrello_3 * Kt_carrelli;
END_IF

IF NOT Alm_Quota_Max_C2_C4 AND NOT Alm_Quota_Min_C2_C4  THEN 
	Pos_Abs_Carrello_2:= Target_Pos_Carrello_2 * Kt_carrelli;
	Pos_Abs_Carrello_4:= Target_Pos_Carrello_4 * Kt_carrelli;
END_IF

IF NOT Alm_Quota_Max_Larg_Bracci AND NOT Alm_Quota_Min_Larg_Bracci  THEN 
	Pos_Abs_Larg_Bracci:= Target_Pos_Larg_Bracci * Kt_Larg_Bracci;
END_IF

IF NOT Alm_Quota_Max_Pinze AND NOT Alm_Quota_Min_Pinze THEN 
	Pos_Abs_Pinza_Sx:= Target_Pos_Pinza_Sx * Kt_Pinze / 3;
	Pos_Abs_Pinza_Dx:= Target_Pos_Pinza_Dx * Kt_Pinze / 3;
END_IF

//esecuzione del comando di set position degli assi all'avvio
//carrello 1
IF C1_attivo AND C1_setpos AND NOT C1_setpos_avviato AND NOT BusySPos_Carrello1 AND NOT Done_SetPosition_C1 AND NOT C1_setpos_eseguito THEN
	Position_Carrello_1:= Pos_Abs_Carrello_1;
	SetPosition_Carrello_1:= TRUE;
	Ref_Carrello_1:= FALSE;		
	C1_setpos_avviato:= TRUE;
END_IF
IF C1_attivo AND C1_setpos AND C1_setpos_avviato THEN
	IF 	Done_SetPosition_C1 THEN
		SetPosition_Carrello_1:= FALSE;
		C1_setpos_avviato:= FALSE;
		Ref_Carrello_1:=TRUE;
	END_IF
END_IF
C1_setpos_eseguito:= (Done_SetPosition_C1 OR C1_setpos_eseguito) AND C1_setpos;

//carrello 2
IF C2_attivo AND C2_setpos AND NOT C2_setpos_avviato AND NOT BusySPos_Carrello2 AND NOT Done_SetPosition_C2 AND NOT C2_setpos_eseguito THEN
	Position_Carrello_2:= Pos_Abs_Carrello_2;
	SetPosition_Carrello_2:= TRUE;
	Ref_Carrello_2:= FALSE;		
	C2_setpos_avviato:= TRUE;
END_IF
IF C2_attivo AND C2_setpos AND C2_setpos_avviato THEN
	IF 	Done_SetPosition_C2 THEN
		SetPosition_Carrello_2:= FALSE;
		C2_setpos_avviato:= FALSE;
		Ref_Carrello_2:=TRUE;
	END_IF
END_IF
C2_setpos_eseguito:= (Done_SetPosition_C2 OR C2_setpos_eseguito) AND C2_setpos;

//carrello 3
IF C3_attivo AND C3_setpos AND NOT C3_setpos_avviato AND NOT BusySPos_Carrello3 AND NOT Done_SetPosition_C3 AND NOT C3_setpos_eseguito THEN
	Position_Carrello_3:= Pos_Abs_Carrello_3;
	SetPosition_Carrello_3:= TRUE;
	Ref_Carrello_3:= FALSE;		
	C3_setpos_avviato:= TRUE;
END_IF
IF C3_attivo AND C3_setpos AND C3_setpos_avviato THEN
	IF 	Done_SetPosition_C3 THEN
		SetPosition_Carrello_3:= FALSE;
		C3_setpos_avviato:= FALSE;
		Ref_Carrello_3:=TRUE;
	END_IF
END_IF
C3_setpos_eseguito:= (Done_SetPosition_C3 OR C3_setpos_eseguito) AND C3_setpos;

//carrello 4
IF C4_attivo AND C4_setpos AND NOT C4_setpos_avviato AND NOT BusySPos_Carrello4 AND NOT Done_SetPosition_C4 AND NOT C4_setpos_eseguito THEN
	Position_Carrello_4:= Pos_Abs_Carrello_4;
	SetPosition_Carrello_4:= TRUE;
	Ref_Carrello_4:= FALSE;		
	C4_setpos_avviato:= TRUE;
END_IF
IF C4_attivo AND C4_setpos AND C4_setpos_avviato THEN
	IF 	Done_SetPosition_C4 THEN
		SetPosition_Carrello_4:= FALSE;
		C4_setpos_avviato:= FALSE;
		Ref_Carrello_4:=TRUE;
	END_IF
END_IF
C4_setpos_eseguito:= (Done_SetPosition_C4 OR C4_setpos_eseguito) AND C4_setpos;

//larghezza bracci
IF Larg_Bracci_attivo AND Larg_Bracci_setpos AND NOT Larg_Bracci_setpos_avviato AND NOT BusySPos_Larg_Bracci AND
			NOT Done_SetPosition_Larg_Bracci AND NOT Larg_Bracci_setpos_eseguito THEN
	Position_Larg_Bracci:= Pos_Abs_Larg_Bracci;
	SetPosition_Larg_Bracci:= TRUE;
	Ref_Larg_Bracci:= FALSE;	
	Larg_Bracci_setpos_avviato:= TRUE;
END_IF
IF Larg_Bracci_attivo AND Larg_Bracci_setpos AND Larg_Bracci_setpos_avviato THEN
	IF Done_SetPosition_Larg_Bracci THEN
		SetPosition_Larg_Bracci:= FALSE;
		Larg_Bracci_setpos_avviato:= FALSE;
		Ref_Larg_Bracci:= TRUE;	
	END_IF
END_IF
Larg_Bracci_setpos_eseguito:= (Done_SetPosition_Larg_Bracci OR Larg_Bracci_setpos_eseguito) AND Larg_Bracci_setpos;

//pinza sinistra
IF Pinza_Sx_attivo AND Pinza_Sx_setpos AND NOT Pinza_Sx_setpos_avviato AND NOT BusySPos_Pinza_Sx AND 
			NOT Done_SetPosition_Pinza_Sx AND NOT Pinza_Sx_setpos_eseguito THEN
	Position_Pinza_Sx:= Pos_Abs_Pinza_Sx;
	SetPosition_Pinza_Sx:= TRUE;
	Ref_Pinza_Sx:= FALSE;	
	Pinza_Sx_setpos_avviato:= TRUE;
END_IF
IF Pinza_Sx_attivo AND Pinza_Sx_setpos AND Pinza_Sx_setpos_avviato THEN
	IF Done_SetPosition_Pinza_Sx THEN
		SetPosition_Pinza_Sx:= FALSE;
		Pinza_Sx_setpos_avviato:= FALSE;
		Ref_Pinza_Sx:= TRUE;	
	END_IF
END_IF
Pinza_Sx_setpos_eseguito:= (Done_SetPosition_Pinza_Sx OR Pinza_Sx_setpos_eseguito) AND Pinza_Sx_setpos;

//pinza destra
IF Pinza_Dx_attivo AND Pinza_Dx_setpos AND NOT Pinza_Dx_setpos_avviato AND NOT BusySPos_Pinza_Dx AND 
			NOT Done_SetPosition_Pinza_Dx AND NOT Pinza_Dx_setpos_eseguito THEN
	Position_Pinza_Dx:= Pos_Abs_Pinza_Dx;
	SetPosition_Pinza_Dx:= TRUE;
	Ref_Pinza_Dx:= FALSE;	
	Pinza_Dx_setpos_avviato:= TRUE;
END_IF
IF Pinza_Dx_attivo AND Pinza_Dx_setpos AND Pinza_Dx_setpos_avviato THEN
	IF Done_SetPosition_Pinza_Dx THEN
		SetPosition_Pinza_Dx:= FALSE;
		Pinza_Dx_setpos_avviato:= FALSE;
		Ref_Pinza_Dx:= TRUE;	
	END_IF
END_IF
Pinza_Dx_setpos_eseguito:= (Done_SetPosition_Pinza_Dx OR Pinza_Dx_setpos_eseguito) AND Pinza_Dx_setpos;

//esecuzione del comando di home 
//carrello 1
IF C1_attivo AND C1_home AND NOT C1_home_avviato AND NOT BusyHome_Carrello1 AND NOT DoneHome_Carr1 AND NOT c1_home_eseguito THEN
	Home_Pos_Carrello_1:= Pos_Abs_Carrello_1;
	Home_Carrello_1:= TRUE;
	Ref_Carrello_1:= FALSE;		
	In_Pos_Carrello_1:= FALSE;
	C1_home_avviato:= TRUE;
END_IF
IF C1_attivo AND C1_home AND C1_home_avviato THEN
	IF 	DoneHome_Carr1 THEN
		Home_Carrello_1:= FALSE;
		C1_home_avviato:= FALSE;
		Ref_Carrello_1:=TRUE;
	END_IF
END_IF

c1_home_eseguito:= (DoneHome_Carr1 OR c1_home_eseguito) AND C1_home;

//carrello 2
IF C2_attivo AND C2_home AND NOT C2_home_avviato AND NOT BusyHome_Carrello2 AND NOT DoneHome_Carr2 AND NOT c2_home_eseguito THEN
	Home_Pos_Carrello_2:= Pos_Abs_Carrello_2;
	Home_Carrello_2:= TRUE;
	Ref_Carrello_2:= FALSE;		
	In_Pos_Carrello_2:= FALSE;
	C2_home_avviato:= TRUE;
END_IF
IF C2_attivo AND C2_home AND C2_home_avviato THEN
	IF 	DoneHome_Carr2 THEN
		Home_Carrello_2:= FALSE;
		C2_home_avviato:= FALSE;
		Ref_Carrello_2:= TRUE;
	END_IF
END_IF

c2_home_eseguito:= (DoneHome_Carr2 OR c2_home_eseguito) AND C2_home;

//carrello 3
IF C3_attivo AND C3_home AND NOT C3_home_avviato AND NOT BusyHome_Carrello3 AND NOT DoneHome_Carr3 AND NOT c3_home_eseguito THEN
	Home_Pos_Carrello_3:= Pos_Abs_Carrello_3;
	Home_Carrello_3:= TRUE;
	Ref_Carrello_3:= FALSE;	
	In_Pos_Carrello_3:= FALSE;
	C3_home_avviato:= TRUE;
END_IF
IF C3_attivo AND C3_home AND C3_home_avviato THEN
	IF 	DoneHome_Carr3 THEN
		Home_Carrello_3:= FALSE;
		C3_home_avviato:= FALSE;
		Ref_Carrello_3:= TRUE;	
	END_IF
END_IF

c3_home_eseguito:= (DoneHome_Carr3 OR c3_home_eseguito) AND C3_home;

//carrello 4
IF C4_attivo AND C4_home AND NOT C4_home_avviato AND NOT BusyHome_Carrello4 AND NOT DoneHome_Carr4 AND NOT c4_home_eseguito THEN
	Home_Pos_Carrello_4:= Pos_Abs_Carrello_4;
	Home_Carrello_4:= TRUE;
	Ref_Carrello_4:= FALSE;	
	In_Pos_Carrello_4:= FALSE;
	C4_home_avviato:= TRUE;
END_IF
IF C4_attivo AND C4_home AND C4_home_avviato THEN
	IF 	DoneHome_Carr4 THEN
		Home_Carrello_4:= FALSE;
		C4_home_avviato:= FALSE;
		Ref_Carrello_4:= TRUE;	
	END_IF
END_IF

c4_home_eseguito:= (DoneHome_Carr4 OR c4_home_eseguito) AND C4_home;

//Larg_Bracci
IF Larg_Bracci_attivo AND Larg_Bracci_home AND NOT Larg_Bracci_home_avviato AND NOT BusyHome_Larg_Bracci AND NOT DoneHome_Larg_Bracci AND
			NOT Larg_Bracci_home_eseguito THEN
	Home_Pos_Larg_Bracci:= Pos_Abs_Larg_Bracci;
	Home_Larg_Bracci:= TRUE;
	Ref_Larg_Bracci:= FALSE;	
	In_Pos_Larg_Bracci:= FALSE;
	Larg_Bracci_home_avviato:= TRUE;
END_IF
IF Larg_Bracci_attivo AND Larg_Bracci_home AND Larg_Bracci_home_avviato THEN
	IF DoneHome_Larg_Bracci THEN
		Home_Larg_Bracci:= FALSE;
		Larg_Bracci_home_avviato:= FALSE;
		Ref_Larg_Bracci:= TRUE;	
	END_IF
END_IF

Larg_Bracci_home_eseguito:= (DoneHome_Larg_Bracci OR Larg_Bracci_home_eseguito) AND Larg_Bracci_home;

//pinza sinistra
IF Pinza_Sx_attivo AND Pinza_Sx_home AND NOT Pinza_Sx_home_avviato AND NOT BusyHome_Pinza_Sx AND NOT DoneHome_Pinza_Sx AND
			NOT Pinza_Sx_home_eseguito THEN
	Home_Pos_Pinza_Sx:= Pos_Abs_Pinza_Sx;
	Home_Pinza_Sx:= TRUE;
	Ref_Pinza_Sx:= FALSE;		
	In_Pos_Pinza_Sx:= FALSE;
	Pinza_Sx_home_avviato:= TRUE;
END_IF
IF Pinza_Sx_attivo AND Pinza_Sx_home AND Pinza_Sx_home_avviato THEN
	IF 	DoneHome_Pinza_Sx THEN
		Home_Pinza_Sx:= FALSE;
		Pinza_Sx_home_avviato:= FALSE;
		Ref_Pinza_Sx:= TRUE;	
	END_IF
END_IF

Pinza_Sx_home_eseguito:= (DoneHome_Pinza_Sx OR Pinza_Sx_home_eseguito) AND Pinza_Sx_home;

//pinza destra
IF Pinza_Dx_attivo AND Pinza_Dx_home AND NOT Pinza_Dx_home_avviato AND NOT BusyHome_Pinza_Dx AND NOT DoneHome_Pinza_Dx AND
			NOT Pinza_Dx_home_eseguito THEN
	Home_Pos_Pinza_Dx:= Pos_Abs_Pinza_Dx;
	Home_Pinza_Dx:= TRUE;
	Ref_Pinza_Dx:= FALSE;		
	In_Pos_Pinza_Dx:= FALSE;
	Pinza_Dx_home_avviato:= TRUE;
END_IF
IF Pinza_Dx_attivo AND Pinza_Dx_home AND Pinza_Dx_home_avviato THEN
	IF 	DoneHome_Pinza_Dx THEN
		Home_Pinza_Dx:= FALSE;
		Pinza_Dx_home_avviato:= FALSE;
		Ref_Pinza_Dx:= TRUE;		
	END_IF
END_IF

Pinza_Dx_home_eseguito:= (DoneHome_Pinza_Dx OR Pinza_Dx_home_eseguito) AND Pinza_Dx_home;

//abort della ricerca dell'home carrello 1
IF Home_Carrello_1 AND NOT C1_home THEN
	Home_Carrello_1:= FALSE;
	C1_home_avviato:= FALSE;
	Stop_Carrello_1:= TRUE;
END_IF
T_stop_C1(In:= Stop_Carrello_1, PT:= T#24MS);
IF T_stop_C1.Q THEN
	Stop_Carrello_1:= FALSE;
END_IF

//abort della ricerca dell'home carrello 2
IF Home_Carrello_2 AND NOT C2_home THEN
	Home_Carrello_2:= FALSE;
	C2_home_avviato:= FALSE;
	Stop_Carrello_2:= TRUE;
END_IF
T_stop_C2(In:= Stop_Carrello_2, PT:= T#24MS);
IF T_stop_C2.Q THEN
	Stop_Carrello_2:= FALSE;
END_IF

//abort della ricerca dell'home carrello 3
IF Home_Carrello_3 AND NOT C3_home THEN
	Home_Carrello_3:= FALSE;
	C3_home_avviato:= FALSE;
	Stop_Carrello_3:= TRUE;
END_IF
T_stop_C3(In:= Stop_Carrello_3, PT:= T#24MS);
IF T_stop_C3.Q THEN
	Stop_Carrello_3:= FALSE;
END_IF

//abort della ricerca dell'home carrello 4
IF Home_Carrello_4 AND NOT C4_home THEN
	Home_Carrello_4:= FALSE;
	C4_home_avviato:= FALSE;
	Stop_Carrello_4:= TRUE;
END_IF
T_stop_C4(In:= Stop_Carrello_4, PT:= T#24MS);
IF T_stop_C4.Q THEN
	Stop_Carrello_4:= FALSE;
END_IF

//abort della ricerca dell'home Larghezza Bracci
IF Home_Larg_Bracci AND NOT Larg_Bracci_home THEN
	Home_Larg_Bracci:= FALSE;
	Larg_Bracci_home_avviato:= FALSE;
	Stop_Larg_Bracci:= TRUE;
END_IF
T_stop_Larg_Bracci(In:= Stop_Larg_Bracci, PT:= T#24MS);
IF T_stop_Larg_Bracci.Q THEN
	Stop_Larg_Bracci:= FALSE;
END_IF

//abort della ricerca dell'home pinza sinistra
IF Home_Pinza_Sx AND NOT Pinza_Sx_home THEN
	Home_Pinza_Sx:= FALSE;
	Pinza_Sx_home_avviato:= FALSE;
	Stop_Pinza_Sx:= TRUE;
END_IF
T_stop_Pinza_Sx(In:= Stop_Pinza_Sx, PT:= T#24MS);
IF T_stop_Pinza_Sx.Q THEN
	Stop_Pinza_Sx:= FALSE;
END_IF

//abort della ricerca dell'home pinza destra
IF Home_Pinza_Dx AND NOT Pinza_Dx_home THEN
	Home_Pinza_Dx:= FALSE;
	Pinza_Dx_home_avviato:= FALSE;
	Stop_Pinza_Dx:= TRUE;
END_IF
T_stop_Pinza_Dx(In:= Stop_Pinza_Dx, PT:= T#24MS);
IF T_stop_Pinza_Dx.Q THEN
	Stop_Pinza_Dx:= FALSE;
END_IF

//esecuzione del comando di posizionamento
//Carrello 1
IF C1_attivo AND C1_position AND NOT C1_pos_avviato AND Ref_Carrello_1 AND NOT Done_Abs_Carrello_1 AND NOT c1_pos_eseguito THEN
	Abs_Carrello_1:= TRUE;		//target di posizione già caricato in Position_Carrello_1
	C1_pos_avviato:= TRUE;
	In_Pos_Carrello_1:= FALSE;
END_IF
IF T_avvio_corsa_C1.Q AND Done_Abs_Carrello_1 THEN
	Abs_Carrello_1:= FALSE;	
	C1_pos_avviato:= FALSE;
	In_Pos_Carrello_1:= TRUE;
END_IF
//attesa avviamento effettivo della corsa prima di controllarne l'arrivo
T_avvio_corsa_C1(IN:= C1_pos_avviato, PT:= T#30MS);

c1_pos_eseguito:= (Done_Abs_Carrello_1 OR c1_pos_eseguito) AND C1_position;

//Carrello 2
IF C2_attivo AND C2_position AND NOT C2_pos_avviato AND Ref_Carrello_2 AND NOT Done_Abs_Carrello_2 AND NOT c2_pos_eseguito THEN
	Abs_Carrello_2:= TRUE;		//target di posizione già caricato in Position_Carrello_2
	C2_pos_avviato:= TRUE;
	In_Pos_Carrello_2:= FALSE;
END_IF
IF T_avvio_corsa_C2.Q AND Done_Abs_Carrello_2 THEN
	Abs_Carrello_2:= FALSE;		
	C2_pos_avviato:= FALSE;
	In_Pos_Carrello_2:= TRUE;
END_IF
//attesa avviamento effettivo della corsa prima di controllarne l'arrivo
T_avvio_corsa_C2(IN:= C2_pos_avviato, PT:= T#30MS);

c2_pos_eseguito:= (Done_Abs_Carrello_2 OR c2_pos_eseguito) AND C2_position;

//Carrello 3
IF C3_attivo AND C3_position AND NOT C3_pos_avviato AND Ref_Carrello_3 AND NOT Done_Abs_Carrello_3 AND NOT c3_pos_eseguito THEN
	Abs_Carrello_3:= TRUE;		//target di posizione già caricato in Position_Carrello_3
	C3_pos_avviato:= TRUE;
	In_Pos_Carrello_3:= FALSE;
END_IF
IF T_avvio_corsa_C3.Q AND Done_Abs_Carrello_3 THEN
	Abs_Carrello_3:= FALSE;	
	C3_pos_avviato:= FALSE;
	In_Pos_Carrello_3:= TRUE;
END_IF
//attesa avviamento effettivo della corsa prima di controllarne l'arrivo
T_avvio_corsa_C3(IN:= C3_pos_avviato, PT:= T#30MS);

c3_pos_eseguito:= (Done_Abs_Carrello_3 OR c3_pos_eseguito) AND C3_position;

//Carrello 4
IF C4_attivo AND C4_position AND NOT C4_pos_avviato AND Ref_Carrello_4 AND NOT Done_Abs_Carrello_4 AND NOT c4_pos_eseguito THEN
	Abs_Carrello_4:= TRUE;		//target di posizione già caricato in Position_Carrello_4
	C4_pos_avviato:= TRUE;
	In_Pos_Carrello_4:= FALSE;
END_IF
IF T_avvio_corsa_C4.Q AND Done_Abs_Carrello_4 THEN
	Abs_Carrello_4:= FALSE;	
	C4_pos_avviato:= FALSE;
	In_Pos_Carrello_4:= TRUE;
END_IF
//attesa avviamento effettivo della corsa prima di controllarne l'arrivo
T_avvio_corsa_C4(IN:= C4_pos_avviato, PT:= T#30MS);

c4_pos_eseguito:= (Done_Abs_Carrello_4 OR c4_pos_eseguito) AND C4_position;

//Larghezza Bracci
IF Larg_Bracci_attivo AND Larg_Bracci_position AND NOT Larg_Bracci_pos_avviato AND Ref_Larg_Bracci AND NOT Done_Abs_Larg_Bracci AND
			NOT Larg_Bracci_pos_eseguito THEN
	Abs_Larg_Bracci:= TRUE;		//target di posizione già caricato in Position_Larg_Bracci
	Larg_Bracci_pos_avviato:= TRUE;
	In_Pos_Larg_Bracci:= FALSE;
END_IF
IF T_avvio_corsa_Larg_Bracci.Q AND Done_Abs_Larg_Bracci THEN
	Abs_Larg_Bracci:= FALSE;
	Larg_Bracci_pos_avviato:= FALSE;
	In_Pos_Larg_Bracci:= TRUE;
END_IF
//attesa avviamento effettivo della corsa prima di controllarne l'arrivo
T_avvio_corsa_Larg_Bracci(IN:= Larg_Bracci_pos_avviato, PT:= T#30MS);

Larg_Bracci_pos_eseguito:= (Done_Abs_Larg_Bracci OR Larg_Bracci_pos_eseguito) AND Larg_Bracci_position;

//Pinza sinistra
IF Pinza_Sx_attivo AND Pinza_Sx_position AND NOT Pinza_Sx_pos_avviato AND Ref_Pinza_Sx AND NOT Done_Abs_Pinza_Sx AND NOT Pinza_Sx_pos_eseguito THEN
	Abs_Pinza_Sx:= TRUE;		//target di posizione già caricato in Pos_Abs_Pinza_Sx
	Pinza_Sx_pos_avviato:= TRUE;
	In_Pos_Pinza_Sx:= FALSE;
END_IF
IF T_avvio_corsa_Pinza_Sx.Q AND Done_Abs_Pinza_Sx THEN
	Abs_Pinza_Sx:= FALSE;	
	Pinza_Sx_pos_avviato:= FALSE;
	In_Pos_Pinza_Sx:= TRUE;
END_IF
//attesa avviamento effettivo della corsa prima di controllarne l'arrivo
T_avvio_corsa_Pinza_Sx(IN:= Pinza_Sx_pos_avviato, PT:= T#30MS);

Pinza_Sx_pos_eseguito:= (Done_Abs_Pinza_Sx OR Pinza_Sx_pos_eseguito) AND Pinza_Sx_position;

//Pinza destra
IF Pinza_Dx_attivo AND Pinza_Dx_position AND NOT Pinza_Dx_pos_avviato AND Ref_Pinza_Dx AND NOT Done_Abs_Pinza_Dx AND NOT Pinza_Dx_pos_eseguito THEN
	Abs_Pinza_Dx:= TRUE;		//target di posizione già caricato in Pos_Abs_Pinza_Dx
	Pinza_Dx_pos_avviato:= TRUE;
	In_Pos_Pinza_Dx:= FALSE;
END_IF
IF T_avvio_corsa_Pinza_Dx.Q AND Done_Abs_Pinza_Dx THEN
	Abs_Pinza_Dx:= FALSE;	
	Pinza_Dx_pos_avviato:= FALSE;
	In_Pos_Pinza_Dx:= TRUE;
END_IF
//attesa avviamento effettivo della corsa prima di controllarne l'arrivo
T_avvio_corsa_Pinza_Dx(IN:= Pinza_Dx_pos_avviato, PT:= T#30MS);

Pinza_Dx_pos_eseguito:= (Done_Abs_Pinza_Dx OR Pinza_Dx_pos_eseguito) AND Pinza_Dx_position;

//esecuzione del comando di jog come inseguimento del volantino
//Carrelli
IF sample_clock THEN
	IF Unita_10X OR DI_Unita_10X THEN
		Delta_encvol:=Delta_encvol*10;
		END_IF
	IF C1_attivo AND C1_jog AND Ref_Carrello_1 THEN
		Distance_Add_Carrello_1:= Delta_encvol * Kt_carrelli; //assumo che l'encoder fornisca 100 imp./mm
		IF Delta_encvol < 0 OR NOT %IX55.3 THEN
			Add_Carrello_1:= TRUE;		
		END_IF
	END_IF
	IF C2_attivo AND C2_jog AND Ref_Carrello_2  THEN
		Distance_Add_Carrello_2:= Delta_encvol * Kt_carrelli; //assumo che l'encoder fornisca 100 imp./mm
		IF Delta_encvol < 0 OR NOT %IX63.3 THEN
			Add_Carrello_2:= TRUE;		
		END_IF
	END_IF
	IF C3_attivo AND C3_jog AND Ref_Carrello_3 THEN
		Distance_Add_Carrello_3:= Delta_encvol * Kt_carrelli; //assumo che l'encoder fornisca 100 imp./mm
		IF Delta_encvol < 0 OR NOT %IX71.3 THEN
			Add_Carrello_3:= TRUE;		
		END_IF
	END_IF
	IF C4_attivo AND C4_jog AND Ref_Carrello_4 THEN
		Distance_Add_Carrello_4:= Delta_encvol * Kt_carrelli; //assumo che l'encoder fornisca 100 imp./mm
		IF Delta_encvol < 0 OR NOT %IX79.3 THEN
			Add_Carrello_4:= TRUE;		
		END_IF
	END_IF
END_IF

T_exe_add_C1(In:= Add_Carrello_1, PT:= T#16MS);
IF T_exe_add_C1.Q THEN
	Add_Carrello_1:= FALSE;	
END_IF
T_exe_add_C2(In:= Add_Carrello_2, PT:= T#16MS);
IF T_exe_add_C2.Q THEN
	Add_Carrello_2:= FALSE;	
END_IF
T_exe_add_C3(In:= Add_Carrello_3, PT:= T#16MS);
IF T_exe_add_C3.Q THEN
	Add_Carrello_3:= FALSE;	
END_IF
T_exe_add_C4(In:= Add_Carrello_4, PT:= T#16MS);
IF T_exe_add_C4.Q THEN
	Add_Carrello_4:= FALSE;	
END_IF

//esecuzione del comando di jog come inseguimento del volantino
//Larghezza Bracci
IF sample_clock THEN
	IF Unita_10X OR DI_Unita_10X THEN
		Delta_encvol:=Delta_encvol*10;
	END_IF
	IF Larg_Bracci_attivo AND Larg_Bracci_jog AND Ref_Larg_Bracci THEN
		Distance_Add_Larg_Bracci:= Delta_encvol * Kt_Larg_Bracci; //assumo che l'encoder fornisca 100 imp./mm
		IF Delta_encvol < 0 OR NOT %IX87.3 THEN
			Add_Larg_Bracci:= TRUE;		
		END_IF
	END_IF
END_IF
	
T_exe_add_Larg_Bracci(In:= Add_Larg_Bracci, PT:= T#16MS);
IF T_exe_add_Larg_Bracci.Q THEN
	Add_Larg_Bracci:= FALSE;	
END_IF

//esecuzione del comando di jog come inseguimento del volantino
//Pinze
IF sample_clock THEN
	IF Unita_10X OR DI_Unita_10X THEN
		Delta_encvol:=Delta_encvol*10;
	END_IF
	IF Pinza_Sx_attivo AND Pinza_Sx_jog AND Ref_Pinza_Sx THEN
		Distance_Add_Pinza_Sx:= Delta_encvol * Kt_Pinze / 3; //assumo che l'encoder fornisca 100 imp./mm
		IF Delta_encvol < 0 OR NOT %IX95.3 THEN
			Add_Pinza_Sx:= TRUE;		
		END_IF
	END_IF	
	IF Pinza_Dx_attivo AND Pinza_Dx_jog AND Ref_Pinza_Dx THEN
		Distance_Add_Pinza_Dx:= Delta_encvol * Kt_Pinze / 3; //assumo che l'encoder fornisca 100 imp./mm
		IF Delta_encvol < 0 OR NOT %IX103.3 THEN
			Add_Pinza_Dx:= TRUE;		
		END_IF
	END_IF
END_IF
	
T_exe_add_Pinza_Sx(In:= Add_Pinza_Sx, PT:= T#16MS);
IF T_exe_add_Pinza_Sx.Q THEN
	Add_Pinza_Sx:= FALSE;	
END_IF

T_exe_add_Pinza_Dx(In:= Add_Pinza_Dx, PT:= T#16MS);
IF T_exe_add_Pinza_Dx.Q THEN
	Add_Pinza_Dx:= FALSE;	
END_IF

(*
//SetPosition in caso di Power Failure
IF Flag_SPos_Master_C1 AND NOT Done_SetPosition_C1 THEN
	Position_Carrello_1:= Target_Pos_Carrello_1;
	SetPosition_Carrello_1:=TRUE;
	Flag_SPos_Slave_C1:=FALSE;
END_IF

IF Flag_SPos_Master_C2 AND NOT Done_SetPosition_C2 THEN
	Position_Carrello_2:= Target_Pos_Carrello_2;
	SetPosition_Carrello_2:=TRUE;
	Flag_SPos_Slave_C2:=FALSE;
END_IF

IF Flag_SPos_Master_C3 AND NOT Done_SetPosition_C3 THEN
	Position_Carrello_3:= Target_Pos_Carrello_3;
	SetPosition_Carrello_3:=TRUE;
	Flag_SPos_Slave_C3:=FALSE;
END_IF

IF Flag_SPos_Master_C4 AND NOT Done_SetPosition_C4 THEN
	Position_Carrello_4:= Target_Pos_Carrello_4;
	SetPosition_Carrello_4:=TRUE;
	Flag_SPos_Slave_C4:=FALSE;
END_IF

IF Flag_SPos_Master_Bracci AND NOT Done_SetPosition_Larg_Bracci THEN
	Position_Larg_Bracci:= Target_Pos_Larg_Bracci;
	SetPosition_Larg_Bracci:=TRUE;
	Flag_SPos_Slave_Bracci:=FALSE;
END_IF

IF Flag_SPos_Master_Pinza_Sx AND NOT Done_SetPosition_Pinza_Sx THEN
	Position_Pinza_Sx:= Target_Pos_Pinza_Sx;
	SetPosition_Pinza_Sx:=TRUE;
	Flag_SPos_Slave_Pinza_Sx:=FALSE;
END_IF

IF Flag_SPos_Master_Pinza_Dx AND NOT Done_SetPosition_Pinza_Dx THEN
	Position_Pinza_Dx:= Target_Pos_Pinza_Dx;
	SetPosition_Pinza_Dx:=TRUE;
	Flag_SPos_Slave_Pinza_Dx:=FALSE;
END_IF
*)

//Reset Setposition
IF (SetPosition_Carrello_1 OR C1_setpos_avviato) AND (NOT C1_attivo OR NOT C1_setpos) THEN
	SetPosition_Carrello_1:=FALSE;
	C1_setpos_avviato:= FALSE;
END_IF

IF (SetPosition_Carrello_2 OR C2_setpos_avviato) AND (NOT C2_attivo OR NOT C2_setpos) THEN
	SetPosition_Carrello_2:=FALSE;
	C2_setpos_avviato:= FALSE;
END_IF

IF (SetPosition_Carrello_3 OR C3_setpos_avviato) AND (NOT C3_attivo OR NOT C3_setpos) THEN
	SetPosition_Carrello_3:=FALSE;
	C3_setpos_avviato:= FALSE;
END_IF

IF (SetPosition_Carrello_4 OR C4_setpos_avviato) AND (NOT C4_attivo OR NOT C4_setpos) THEN
	SetPosition_Carrello_4:=FALSE;
	C4_setpos_avviato:= FALSE;
END_IF

IF (SetPosition_Larg_Bracci OR Larg_Bracci_setpos_avviato) AND (NOT Larg_Bracci_attivo OR NOT Larg_Bracci_setpos) THEN
	SetPosition_Larg_Bracci:=FALSE;
	Larg_bracci_setpos_avviato:= FALSE;
END_IF

IF (SetPosition_Pinza_Sx OR Pinza_Sx_setpos_avviato) AND (NOT Pinza_Sx_attivo OR NOT Pinza_Sx_setpos) THEN
	SetPosition_Pinza_Sx:=FALSE;
	Pinza_Sx_setpos_avviato:=FALSE;
END_IF

IF (SetPosition_Pinza_Dx OR Pinza_Dx_setpos_avviato) AND (NOT Pinza_Dx_attivo OR NOT Pinza_Dx_setpos) THEN
	SetPosition_Pinza_Dx:=FALSE;
	Pinza_Dx_setpos_avviato:=FALSE;
END_IF

//Verifica dell'abort dei comandi

F_C1_home(clk:=C1_home);
F_C2_home(clk:=C2_home);
F_C3_home(clk:=C3_home);
F_C4_home(clk:=C4_home);
F_C1_pos(clk:=C1_position);
F_C2_pos(clk:=C2_position);
F_C3_pos(clk:=C3_position);
F_C4_pos(clk:=C4_position);

F_Larg_Bracci_Home(clk:=Larg_Bracci_home);
F_Pinza_Sx_Home(clk:=Pinza_Sx_home);
F_Pinza_Dx_Home(clk:=Pinza_Dx_home);
F_Larg_Bracci_Pos(clk:=Larg_Bracci_position);
F_Pinxa_Sx_Pos(clk:=Pinza_Sx_position);
F_Pinxa_Dx_Pos(clk:=Pinza_Dx_position);

//reset assi in errore
Reset_Carrello_1:= Error_Carrello_1 AND Cancella_allarmi;
Reset_Carrello_2:= Error_Carrello_2 AND Cancella_allarmi;
Reset_Carrello_3:= Error_Carrello_3 AND Cancella_allarmi;
Reset_Carrello_4:= Error_Carrello_4 AND Cancella_allarmi;
Reset_Larg_Bracci:= Error_Larg_Bracci AND Cancella_allarmi;
Reset_Pinza_Sx:= Error_Pinza_Sx AND Cancella_allarmi;
Reset_Pinza_Dx:= Error_Pinza_Dx AND Cancella_allarmi;

IF Reset_Carrello_1 OR F_C1_home.Q AND NOT Ref_Carrello_1 OR F_C1_pos.Q AND NOT In_Pos_Carrello_1 THEN
	Home_Carrello_1:= FALSE;
	Abs_Carrello_1:= FALSE;
	C1_home_avviato:= FALSE;
	C1_Pos_avviato:= FALSE;
END_IF
IF Reset_Carrello_2 OR F_C2_home.Q AND NOT Ref_Carrello_2 OR F_C2_pos.Q AND NOT In_Pos_Carrello_2 THEN
	Home_Carrello_2:= FALSE;
	Abs_Carrello_2:= FALSE;
	C2_home_avviato:= FALSE;
	C2_Pos_avviato:= FALSE;
END_IF
IF Reset_Carrello_3 OR F_C3_home.Q AND NOT Ref_Carrello_3 OR F_C3_pos.Q AND NOT In_Pos_Carrello_3 THEN
	Home_Carrello_3:= FALSE;
	Abs_Carrello_3:= FALSE;
	C3_home_avviato:= FALSE;
	C3_Pos_avviato:= FALSE;
END_IF
IF Reset_Carrello_4 OR F_C4_home.Q AND NOT Ref_Carrello_4 OR F_C4_pos.Q AND NOT In_Pos_Carrello_4 THEN
	Home_Carrello_4:= FALSE;
	Abs_Carrello_4:= FALSE;
	C4_home_avviato:= FALSE;
	C4_Pos_avviato:= FALSE;
END_IF
IF Reset_Larg_Bracci OR F_Larg_Bracci_home.Q AND NOT Ref_Larg_Bracci OR F_Larg_Bracci_pos.Q AND NOT In_Pos_Larg_Bracci THEN
	Home_Larg_Bracci:= FALSE;
	Abs_Larg_Bracci:= FALSE;
	Larg_Bracci_home_avviato:= FALSE;
	Larg_Bracci_Pos_avviato:= FALSE;
END_IF
IF Reset_Pinza_Sx OR F_Pinza_Sx_home.Q AND NOT Ref_Pinza_Sx OR F_Pinxa_Sx_Pos.Q AND NOT In_Pos_Pinza_Sx THEN
	Home_Pinza_Sx:= FALSE;
	Abs_Pinza_Sx:= FALSE;
	Pinza_Sx_home_avviato:= FALSE;
	Pinza_Sx_Pos_avviato:= FALSE;
END_IF
IF Reset_Pinza_Dx OR F_Pinza_Dx_home.Q AND NOT Ref_Pinza_Dx OR F_Pinxa_Dx_Pos.Q AND NOT In_Pos_Pinza_Dx THEN
	Home_Pinza_Dx:= FALSE;
	Abs_Pinza_Dx:= FALSE;
	Pinza_Dx_home_avviato:= FALSE;
	Pinza_Dx_Pos_avviato:= FALSE;
END_IF

END_PROGRAM

// MyController/Application/Programma/P7_Allarmi
PROGRAM P7_Allarmi
VAR
END_VAR

//Allarmi su eventuale errore di ricezione di una posizione target
//carrello 1 o 3
(*IF Target_Pos_Carrello_1 <= M241_Lungh_Min_Scat OR
	Target_Pos_Carrello_3 <= M241_Lungh_Min_Scat THEN 
	Alm_Quota_Min_C1_C3:= TRUE; 
ELSE
	Alm_Quota_Min_C1_C3:= FALSE;
END_IF*)
IF Target_Pos_Carrello_1 > M241_Lungh_Max_Scat OR
	Target_Pos_Carrello_3 > M241_Lungh_Max_Scat THEN 
	Alm_Quota_Max_C1_C3:= TRUE; 
ELSE
	Alm_Quota_Max_C1_C3:= FALSE;
END_IF
//carrello 2 o 4		
(*IF Target_Pos_Carrello_2 < M241_Largh_Min_Scat OR
	Target_Pos_Carrello_4 < M241_Largh_Min_Scat THEN 
	Alm_Quota_Min_C2_C4:= TRUE; 
ELSE
	Alm_Quota_Min_C2_C4:= FALSE;
END_IF*)
IF Target_Pos_Carrello_2 > M241_Largh_Max_Scat OR
	Target_Pos_Carrello_4 > M241_Largh_Max_Scat THEN 
	Alm_Quota_Max_C2_C4:= TRUE; 
ELSE
	Alm_Quota_Max_C2_C4:= FALSE;
END_IF

//Larg_Bracci						
(*IF Target_Pos_Larg_Bracci < M241_Lungh_Min_Scat THEN 
	Alm_Quota_Min_Larg_Bracci:= TRUE; 
ELSE
	Alm_Quota_Min_Larg_Bracci:= FALSE;
END_IF*)
IF Target_Pos_Larg_Bracci > M241_Lungh_Max_Scat THEN 
	Alm_Quota_Max_Larg_Bracci:= TRUE; 
ELSE
	Alm_Quota_Max_Larg_Bracci:= FALSE;
END_IF

//Pinze 1 o 2								
(*IF Target_Pos_Pinza_Sx < M241_Largh_Min_Scat OR
 	Target_Pos_Pinza_Dx < M241_Largh_Min_Scat THEN 
	Alm_Quota_Min_Pinze:= TRUE; 
ELSE
	Alm_Quota_Min_Pinze:= FALSE;
END_IF*)
IF Target_Pos_Pinza_Sx > M241_Largh_Max_Scat OR
	Target_Pos_Pinza_Dx > M241_Largh_Max_Scat THEN 
	Alm_Quota_Max_Pinze:= TRUE; 
ELSE
	Alm_Quota_Max_Pinze:= FALSE;
END_IF

END_PROGRAM

// MyController/Application/Programma/P9_Slave_to_master
PROGRAM P9_Slave_to_master
VAR
END_VAR

Fault_Carrello_1:= ErrorID_Carrello_1;
Fault_Carrello_2:= ErrorID_Carrello_2;
Fault_Carrello_3:= ErrorID_Carrello_3;
Fault_Carrello_4:= ErrorID_Carrello_4;
Fault_Larg_Bracci:= ErrorID_Larg_Bracci;
Fault_Pinza_Sx:= ErrorID_Pinza_Sx;
Fault_Pinza_Dx:= ErrorID_Pinza_Dx;

Actual_Position_Carrello_1:= DINT_TO_INT(ActPosition_Carrello_1 / Kt_Carrelli);
Actual_Position_Carrello_2:= DINT_TO_INT(ActPosition_Carrello_2 / Kt_Carrelli);
Actual_Position_Carrello_3:= DINT_TO_INT(ActPosition_Carrello_3 / Kt_Carrelli);
Actual_Position_Carrello_4:= DINT_TO_INT(ActPosition_Carrello_4 / Kt_Carrelli);
Actual_Position_Larg_Bracci:= DINT_TO_INT(ActPosition_Larg_Bracci / Kt_Larg_Bracci);
Actual_Position_Pinza_Sx:= DINT_TO_INT(ActPosition_Pinza_Sx * 3 / Kt_Pinze);
Actual_Position_Pinza_Dx:= DINT_TO_INT(ActPosition_Pinza_Dx * 3 / Kt_Pinze);

Actual_Position_Volantino:= DINT_TO_INT(Encoder_Vol);		//100 (400) impulsi a mm (giro)

//assegnazione variabili di scambio in uscita

C1_errore:= Error_Carrello_1 AND modo_regolazioni;
C1_referenced:= Ref_Carrello_1;
C1_done_abs:= c1_pos_eseguito;
C1_done_home:= DoneHome_Carr1;
C1_done_mvadd:= Done_MAdd_Carrello_1;
C1_done_setpos:= C1_setpos_eseguito;
C1_in_position:= In_Pos_Carrello_1;

C2_errore:= Error_Carrello_2 AND modo_regolazioni;
C2_referenced:= Ref_Carrello_2;
C2_done_abs:= c2_pos_eseguito;
C2_done_home:= DoneHome_Carr2;
C2_done_mvadd:= Done_MAdd_Carrello_2;
C2_done_setpos:= C2_setpos_eseguito;
C2_in_position:= In_Pos_Carrello_2;

C3_errore:= Error_Carrello_3 AND modo_regolazioni;
C3_referenced:= Ref_Carrello_3;
C3_done_abs:= c3_pos_eseguito;
C3_done_home:= DoneHome_Carr3;
C3_done_mvadd:= Done_MAdd_Carrello_3;
C3_done_setpos:= C3_setpos_eseguito;
C3_in_position:= In_Pos_Carrello_3;

C4_errore:= Error_Carrello_4 AND modo_regolazioni;
C4_referenced:= Ref_Carrello_4;
C4_done_abs:= c4_pos_eseguito;
C4_done_home:= DoneHome_Carr4;
C4_done_mvadd:= Done_MAdd_Carrello_4;
C4_done_setpos:= C4_setpos_eseguito;
C4_in_position:= In_Pos_Carrello_4;

L_br_errore:= Error_Larg_Bracci AND modo_regolazioni;
L_br_referenced:= Ref_Larg_Bracci;
L_br_done_abs:= Larg_Bracci_pos_eseguito;
L_br_done_home:= DoneHome_Larg_Bracci;
L_br_done_mvadd:= Done_MAdd_Larg_Bracci;
L_br_done_setpos:= Larg_Bracci_setpos_eseguito;
L_br_in_position:= In_Pos_Larg_bracci;

Pinza_Sx_errore:= Error_Pinza_Sx AND modo_regolazioni;
Pinza_Sx_referenced:= Ref_Pinza_Sx;
Pinza_Sx_done_abs:= Pinza_Sx_pos_eseguito;
Pinza_Sx_done_home:= DoneHome_Pinza_Sx;
Pinza_Sx_done_mvadd:= Done_MAdd_Pinza_Sx;
Pinza_Sx_done_setpos:= Pinza_Sx_setpos_eseguito;
Pinza_Sx_in_position:= In_Pos_Pinza_Sx;

Pinza_Dx_errore:= Error_Pinza_Dx AND modo_regolazioni;
Pinza_Dx_referenced:= Ref_Pinza_Dx;
Pinza_Dx_done_abs:= Pinza_Dx_pos_eseguito;
Pinza_Dx_done_home:= DoneHome_Pinza_Dx;
Pinza_Dx_done_mvadd:= Done_MAdd_Pinza_Dx;
Pinza_Dx_done_setpos:= Pinza_Dx_setpos_eseguito;
Pinza_Dx_in_position:= In_Pos_Pinza_Dx;

//Risposta alla query del PLC Master
Reverse_Token:= NOT Token;       //risposta al token
PB_Abil_Vol:= UM_Abil_Vol;			// immagine tasto volantino verso CPU master

END_PROGRAM

// MyController/Application/FB_Steppers
FUNCTION_BLOCK FB_Steppers
VAR_INPUT
	
	i_Power: BOOL;
	i_DriveReady_Power: BOOL;
	i_LimP_Power: BOOL;
	i_LimN_Power: BOOL;
	i_Reset: BOOL;
	i_Stop: BOOL;
	i_Decel_Stop: DINT;
	i_JerkRatio_Stop: INT;
	i_ReadAxisError: BOOL;
	i_Home: BOOL;
	i_Mode_Home: PTO_HOMING_MODE;
	i_Position_Home: DINT;
	i_Direction_Home: MC_DIRECTION;
	i_HighVel_Home: DINT;
	i_LowVel_Home: DINT;
	i_Accel_Home: DINT;
	i_Decel_Home: DINT;
	i_Offset_Home: DINT;
	i_JerkRatio_Home: INT;
	i_MoveAbsolute: BOOL;
	i_Position_MoveAbs: DINT;
	i_Vel_MoveAbs: DINT;
	i_Accel_MoveAbs: DINT;
	i_Decel_MoveAbs: DINT;
	i_BufferMode_MoveAbs: MC_BUFFER_MODE;
	i_JerkRatio_MoveAbs: INT;
	i_MoveRelative: BOOL;
	i_Distance_MoveRelative: DINT;
	i_Vel_MoveRelative: DINT;
	i_Accel_MoveRelative: DINT;
	i_Decel_MoveRelative: DINT;
	i_BufferMode_MoveRelative: MC_BUFFER_MODE;
	i_JerkRatio_MoveRelative: INT;
	i_ReadActualPosition: BOOL;
	i_ReadActualVelocity: BOOL;
	i_SetPosition: BOOL;
	i_Position_SetPosition: DINT;
	i_ReadStatus: BOOL;
END_VAR
VAR_OUTPUT
	q_ErrorId: PTO_ERROR;
	q_StandStill: BOOL;
	q_DoneAbsolute: BOOL;
	q_Done_MoreRelative: BOOL;
	q_Error: BOOL;
	q_ActPosition: DINT;
	q_Busy_Home: BOOL;
	q_Done_SPosition: BOOL;
	q_Busy_Abs: BOOL;
	q_Done_Home: BOOL;
	q_power_status: BOOL;
END_VAR
VAR
	MC_Power_PTO_0: MC_Power_PTO;
	MC_Reset_PTO_0: MC_Reset_PTO;
	MC_Stop_PTO_0: MC_Stop_PTO;
	MC_ReadAxisError_PTO_0: MC_ReadAxisError_PTO;
	MC_Home_PTO_0: MC_Home_PTO;
	MC_MoveAbsolute_PTO_0: MC_MoveAbsolute_PTO;
	MC_MoveRelative_PTO_0: MC_MoveRelative_PTO;
	MC_ReadActualPosition_PTO_0: MC_ReadActualPosition_PTO;
	MC_ReadActualVelocity_PTO_0: MC_ReadActualVelocity_PTO;
	MC_SetPosition_PTO_0: MC_SetPosition_PTO;
	MC_ReadStatus_PTO_0: MC_ReadStatus_PTO;

END_VAR

VAR_IN_OUT
	i_ifAsse: AXIS_REF_PTO;
END_VAR

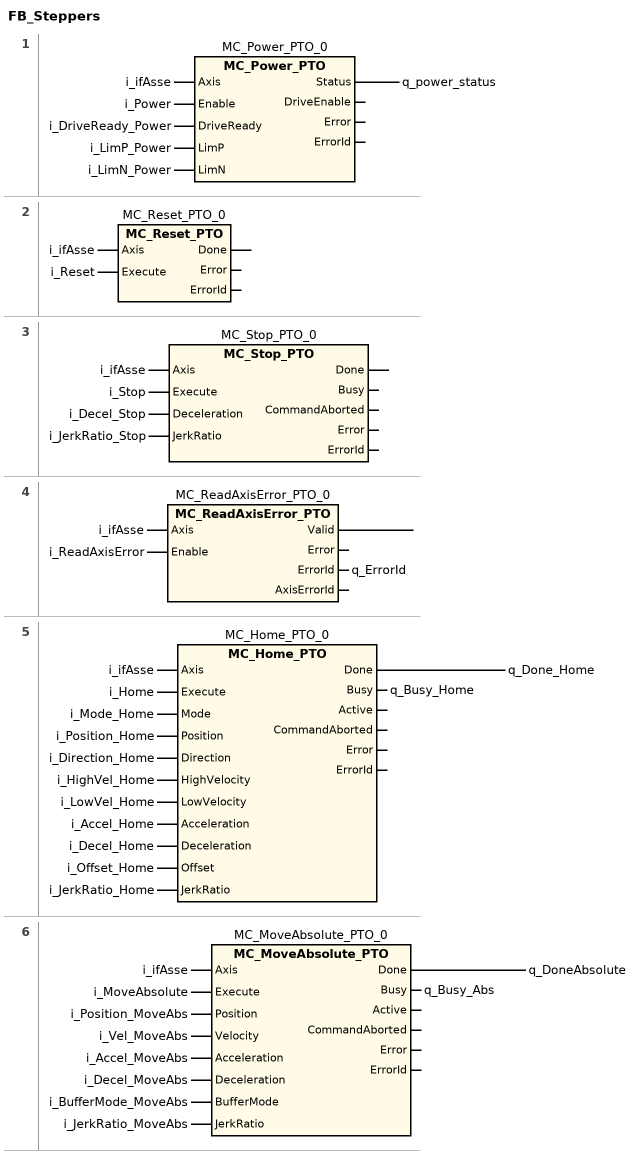
// NETWORK 1
MC_Power_PTO_0(
    Axis := i_ifAsse,
    Enable := i_Power,
    DriveReady := i_DriveReady_Power,
    LimP := i_LimP_Power,
    LimN := i_LimN_Power); // MC_Power_PTO
q_power_status := MC_Power_PTO_0.Status;

// NETWORK 2
MC_Reset_PTO_0(Axis := i_ifAsse, Execute := i_Reset); // MC_Reset_PTO

// NETWORK 3
MC_Stop_PTO_0(
    Axis := i_ifAsse,
    Execute := i_Stop,
    Deceleration := i_Decel_Stop,
    JerkRatio := i_JerkRatio_Stop); // MC_Stop_PTO

// NETWORK 4
MC_ReadAxisError_PTO_0(Axis := i_ifAsse, Enable := i_ReadAxisError, ErrorId => q_ErrorId); // MC_ReadAxisError_PTO

// NETWORK 5
MC_Home_PTO_0(
    Axis := i_ifAsse,
    Execute := i_Home,
    Mode := i_Mode_Home,
    Position := i_Position_Home,
    Direction := i_Direction_Home,
    HighVelocity := i_HighVel_Home,
    LowVelocity := i_LowVel_Home,
    Acceleration := i_Accel_Home,
    Deceleration := i_Decel_Home,
    Offset := i_Offset_Home,
    JerkRatio := i_JerkRatio_Home,
    Busy => q_Busy_Home); // MC_Home_PTO
q_Done_Home := MC_Home_PTO_0.Done;

// NETWORK 6
MC_MoveAbsolute_PTO_0(
    Axis := i_ifAsse,
    Execute := i_MoveAbsolute,
    Position := i_Position_MoveAbs,
    Velocity := i_Vel_MoveAbs,
    Acceleration := i_Accel_MoveAbs,
    Deceleration := i_Decel_MoveAbs,
    BufferMode := i_BufferMode_MoveAbs,
    JerkRatio := i_JerkRatio_MoveAbs,
    Busy => q_Busy_Abs); // MC_MoveAbsolute_PTO
q_DoneAbsolute := MC_MoveAbsolute_PTO_0.Done;

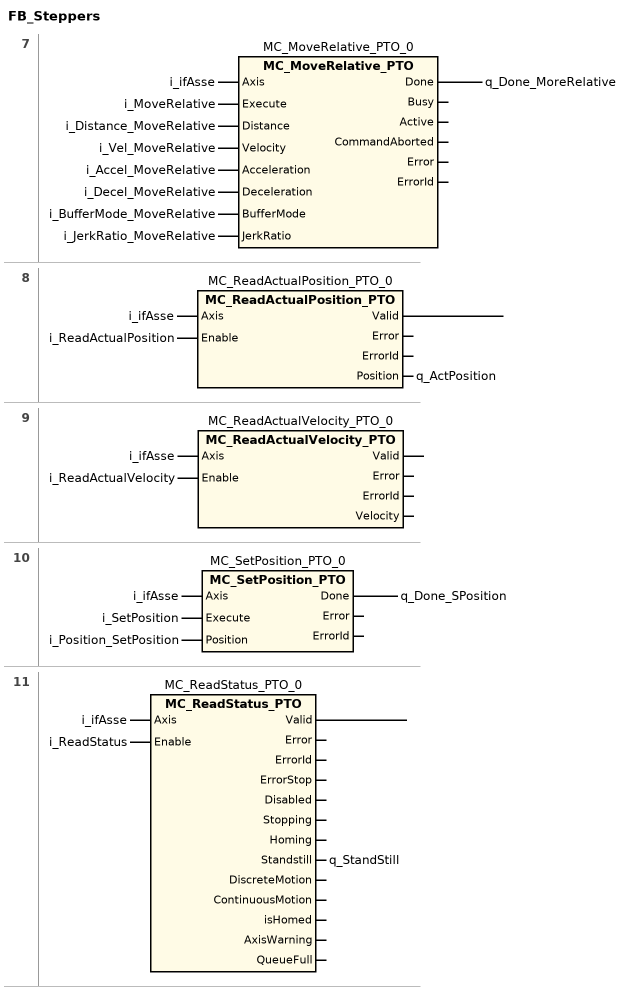
// NETWORK 7
MC_MoveRelative_PTO_0(
    Axis := i_ifAsse,
    Execute := i_MoveRelative,
    Distance := i_Distance_MoveRelative,
    Velocity := i_Vel_MoveRelative,
    Acceleration := i_Accel_MoveRelative,
    Deceleration := i_Decel_MoveRelative,
    BufferMode := i_BufferMode_MoveRelative,
    JerkRatio := i_JerkRatio_MoveRelative); // MC_MoveRelative_PTO
q_Done_MoreRelative := MC_MoveRelative_PTO_0.Done;

// NETWORK 8
MC_ReadActualPosition_PTO_0(Axis := i_ifAsse, Enable := i_ReadActualPosition, Position => q_ActPosition); // MC_ReadActualPosition_PTO

// NETWORK 9
MC_ReadActualVelocity_PTO_0(Axis := i_ifAsse, Enable := i_ReadActualVelocity); // MC_ReadActualVelocity_PTO

// NETWORK 10
MC_SetPosition_PTO_0(Axis := i_ifAsse, Execute := i_SetPosition, Position := i_Position_SetPosition); // MC_SetPosition_PTO
q_Done_SPosition := MC_SetPosition_PTO_0.Done;

// NETWORK 11
MC_ReadStatus_PTO_0(Axis := i_ifAsse, Enable := i_ReadStatus, Standstill => q_StandStill); // MC_ReadStatus_PTO

